C05458=1080.176,351.466,404.288,176.034,28.029,154.818
C05459=1080.171,351.219,404.324,176.031,28.024,154.817
C05460=1080.164,350.972,404.359,176.028,28.019,154.816
C05461=1080.158,350.724,404.394,176.025,28.013,154.815
C05462=1080.153,350.477,404.429,176.022,28.008,154.814
C05463=1080.146,350.229,404.464,176.018,28.002,154.813
C05464=1080.140,349.982,404.500,176.015,27.997,154.812
C05465=1080.134,349.735,404.535,176.012,27.992,154.811
C05466=1080.128,349.487,404.570,176.009,27.987,154.810
C05467=1080.121,349.239,404.605,176.005,27.981,154.809
C05468=1080.116,348.992,404.640,176.002,27.976,154.808
C05469=1080.109,348.745,404.675,175.999,27.971,154.807
C05470=1080.103,348.497,404.710,175.995,27.965,154.807
C05471=1080.097,348.250,404.745,175.992,27.960,154.806
C05472=1080.091,348.002,404.781,175.989,27.955,154.805
C05473=1080.085,347.755,404.815,175.985,27.950,154.804
C05474=1080.079,347.507,404.851,175.982,27.944,154.803
C05475=1080.073,347.259,404.885,175.979,27.939,154.802
C05476=1080.067,347.012,404.920,175.976,27.934,154.801
C05477=1080.061,346.765,404.956,175.973,27.929,154.800
C05478=1080.055,346.518,404.990,175.970,27.924,154.799
C05479=1080.049,346.270,405.025,175.966,27.918,154.798
C05480=1080.043,346.022,405.060,175.963,27.913,154.797
C05481=1080.037,345.775,405.095,175.959,27.908,154.797
C05482=1080.030,345.527,405.130,175.956,27.903,154.796
C05483=1080.025,345.280,405.165,175.953,27.898,154.795
C05484=1080.018,345.032,405.199,175.950,27.893,154.794
C05485=1080.009,344.621,405.257,175.945,27.884,154.793
C05486=1079.998,344.208,405.314,175.939,27.876,154.791
C05487=1079.988,343.795,405.372,175.934,27.867,154.790
C05488=1079.978,343.384,405.430,175.928,27.858,154.788
C05489=1079.972,343.135,405.465,175.925,27.854,154.787
C05490=1079.967,342.888,405.499,175.922,27.848,154.786
C05491=1079.960,342.641,405.534,175.919,27.843,154.786
C05492=1079.954,342.394,405.568,175.916,27.839,154.785
C05493=1079.947,342.146,405.603,175.912,27.833,154.784
C05494=1079.942,341.898,405.637,175.909,27.828,154.783
C05495=1079.936,341.650,405.672,175.906,27.823,154.782
C05496=1079.930,341.403,405.706,175.903,27.818,154.781
C05497=1079.923,341.155,405.741,175.899,27.813,154.781
C05498=1079.917,340.908,405.775,175.896,27.808,154.780
C05499=1079.912,340.661,405.809,175.893,27.803,154.779
C05500=1079.906,340.412,405.844,175.890,27.798,154.778
C05501=1079.900,340.165,405.878,175.887,27.793,154.777
C05502=1079.894,339.917,405.913,175.884,27.788,154.776
C05503=1079.888,339.670,405.947,175.881,27.784,154.775
C05504=1079.882,339.423,405.981,175.877,27.778,154.775
C05505=1079.875,339.175,406.015,175.874,27.773,154.774
C05506=1079.869,338.927,406.049,175.871,27.768,154.773
C05507=1079.864,338.679,406.084,175.867,27.763,154.772
C05508=1079.858,338.432,406.118,175.864,27.758,154.771
C05509=1079.852,338.184,406.152,175.861,27.754,154.770
C05510=1079.846,337.936,406.187,175.858,27.748,154.770
C05511=1079.840,337.689,406.221,175.855,27.744,154.769
C05512=1079.834,337.441,406.254,175.852,27.739,154.768
C05513=1079.828,337.193,406.288,175.849,27.734,154.767
C05514=1079.822,336.946,406.322,175.846,27.729,154.766
C05515=1079.816,336.699,406.357,175.843,27.724,154.766
C05516=1079.809,336.451,406.391,175.839,27.720,154.765
C05517=1079.804,336.203,406.425,175.836,27.715,154.764
C05518=1079.797,335.956,406.458,175.833,27.710,154.763
C05519=1079.791,335.708,406.492,175.830,27.705,154.762
C05520=1079.785,335.461,406.526,175.827,27.700,154.762
C05521=1079.779,335.213,406.560,175.824,27.695,154.761
C05522=1079.773,334.965,406.594,175.821,27.691,154.760
C05523=1079.767,334.717,406.628,175.818,27.685,154.759
C05524=1079.761,334.470,406.662,175.815,27.681,154.758
C05525=1079.756,334.222,406.695,175.811,27.676,154.758
C05526=1079.749,333.974,406.730,175.807,27.671,154.757
C05527=1079.744,333.726,406.763,175.804,27.666,154.756
C05528=1079.737,333.479,406.797,175.801,27.662,154.755
C05529=1079.731,333.232,406.831,175.798,27.656,154.754
C05530=1079.726,332.984,406.864,175.795,27.652,154.754
C05531=1079.719,332.736,406.898,175.792,27.647,154.753
C05532=1079.714,332.488,406.932,175.789,27.642,154.752
C05533=1079.708,332.241,406.966,175.786,27.638,154.751
C05534=1079.702,331.993,406.999,175.783,27.633,154.750
C05535=1079.696,331.746,407.033,175.780,27.628,154.750
C05536=1079.690,331.498,407.066,175.777,27.624,154.749
C05537=1079.679,331.080,407.123,175.772,27.615,154.748
C05538=1079.669,330.662,407.179,175.766,27.608,154.746
C05539=1079.659,330.245,407.235,175.760,27.600,154.745
C05540=1079.648,329.827,407.292,175.756,27.592,154.744
C05541=1079.642,329.579,407.326,175.753,27.588,154.743
C05542=1079.636,329.331,407.358,175.750,27.583,154.742
C05543=1079.630,329.084,407.392,175.746,27.579,154.742
C05544=1079.624,328.836,407.425,175.743,27.574,154.741
C05545=1079.618,328.588,407.458,175.740,27.569,154.740
C05546=1079.612,328.341,407.491,175.737,27.565,154.739
C05547=1079.606,328.092,407.525,175.734,27.560,154.739
C05548=1079.599,327.845,407.558,175.731,27.555,154.738
C05549=1079.594,327.597,407.592,175.728,27.551,154.737
C05550=1079.587,327.350,407.624,175.725,27.546,154.736
C05551=1079.582,327.102,407.658,175.721,27.542,154.736
C05552=1079.575,326.854,407.690,175.718,27.537,154.735
C05553=1079.570,326.606,407.724,175.715,27.533,154.734
C05554=1079.564,326.359,407.757,175.712,27.528,154.733
C05555=1079.558,326.112,407.791,175.709,27.523,154.733
C05556=1079.551,325.863,407.824,175.707,27.519,154.732
C05557=1079.545,325.615,407.857,175.704,27.515,154.731
C05558=1079.539,325.368,407.890,175.700,27.510,154.730
C05559=1079.533,325.120,407.923,175.697,27.506,154.730
C05560=1079.527,324.872,407.956,175.694,27.501,154.729
C05561=1079.521,324.625,407.989,175.691,27.497,154.728
C05562=1079.515,324.377,408.022,175.688,27.492,154.728
C05563=1079.509,324.129,408.055,175.685,27.487,154.727
C05564=1079.503,323.881,408.088,175.682,27.483,154.726
C05565=1079.497,323.633,408.120,175.678,27.478,154.725
C05566=1079.491,323.385,408.153,175.676,27.474,154.725
C05567=1079.486,323.138,408.186,175.673,27.469,154.724
C05568=1079.479,322.890,408.219,175.670,27.465,154.723
C05569=1079.474,322.642,408.252,175.667,27.460,154.723
C05570=1079.467,322.394,408.285,175.664,27.456,154.722
C05571=1079.461,322.147,408.318,175.660,27.451,154.721
C05572=1079.457,321.899,408.350,175.657,27.447,154.720
C05573=1079.450,321.651,408.383,175.654,27.442,154.720
C05574=1079.445,321.404,408.416,175.651,27.438,154.719
C05575=1079.438,321.156,408.449,175.649,27.434,154.718
C05576=1079.432,320.908,408.482,175.646,27.429,154.717
C05577=1079.427,320.660,408.514,175.643,27.425,154.717
C05578=1079.421,320.412,408.547,175.639,27.420,154.716
C05579=1079.414,320.165,408.580,175.636,27.416,154.715
C05580=1079.409,319.916,408.612,175.633,27.411,154.715
C05581=1079.403,319.669,408.645,175.630,27.407,154.714
C05582=1079.397,319.422,408.677,175.628,27.402,154.713
C05583=1079.392,319.173,408.710,175.625,27.398,154.713
C05584=1079.386,318.925,408.743,175.622,27.393,154.712
C05585=1079.379,318.678,408.775,175.618,27.389,154.711
C05586=1079.374,318.430,408.807,175.615,27.384,154.710
C05587=1079.368,318.182,408.840,175.612,27.380,154.710
C05588=1079.362,317.934,408.872,175.610,27.376,154.709
C05589=1079.357,317.723,408.901,175.607,27.372,154.708
C05590=1079.353,317.510,408.928,175.605,27.368,154.708
C05591=1079.347,317.297,408.956,175.602,27.364,154.707
C05592=1079.342,317.086,408.985,175.599,27.360,154.707
C05593=1079.337,316.874,409.012,175.597,27.356,154.706
C05594=1079.332,316.662,409.039,175.594,27.353,154.705
C05595=1079.328,316.449,409.067,175.592,27.349,154.705
C05596=1079.323,316.238,409.095,175.589,27.345,154.704
C05597=1079.317,315.989,409.127,175.587,27.341,154.703
C05598=1079.311,315.741,409.159,175.584,27.337,154.703
C05599=1079.306,315.494,409.192,175.580,27.332,154.702
C05600=1079.300,315.246,409.224,175.577,27.327,154.701
C05601=1079.294,314.998,409.257,175.574,27.323,154.701
C05602=1079.288,314.751,409.289,175.572,27.319,154.700
C05603=1079.282,314.502,409.321,175.569,27.314,154.699
C05604=1079.276,314.255,409.354,175.566,27.310,154.699
C05605=1079.270,314.007,409.386,175.562,27.306,154.698
C05606=1079.264,313.758,409.418,175.559,27.302,154.697
C05607=1079.258,313.511,409.449,175.556,27.297,154.697
C05608=1079.251,313.264,409.481,175.554,27.293,154.696
C05609=1079.245,313.015,409.513,175.551,27.289,154.695
C05610=1079.239,312.767,409.545,175.548,27.285,154.695
C05611=1079.233,312.519,409.578,175.544,27.281,154.694
C05612=1079.228,312.272,409.609,175.541,27.276,154.694
C05613=1079.221,312.024,409.641,175.539,27.272,154.693
C05614=1079.215,311.776,409.673,175.536,27.268,154.692
C05615=1079.210,311.529,409.705,175.533,27.264,154.692
C05616=1079.204,311.280,409.737,175.530,27.260,154.691
C05617=1079.198,311.032,409.769,175.527,27.256,154.690
C05618=1079.191,310.784,409.800,175.524,27.251,154.690
C05619=1079.186,310.537,409.832,175.521,27.247,154.689
C05620=1079.180,310.288,409.864,175.518,27.243,154.688
C05621=1079.174,310.040,409.896,175.515,27.238,154.688
C05622=1079.168,309.793,409.927,175.512,27.234,154.687
C05623=1079.162,309.545,409.959,175.509,27.230,154.686
C05624=1079.156,309.297,409.991,175.506,27.226,154.686
C05625=1079.150,309.049,410.023,175.503,27.222,154.685
C05626=1079.143,308.801,410.054,175.501,27.218,154.684
C05627=1079.138,308.554,410.086,175.498,27.213,154.684
C05628=1079.132,308.305,410.118,175.494,27.209,154.683
C05629=1079.127,308.058,410.150,175.491,27.205,154.682
C05630=1079.120,307.810,410.181,175.488,27.201,154.682
C05631=1079.114,307.562,410.213,175.486,27.197,154.681
C05632=1079.109,307.314,410.245,175.483,27.193,154.681
C05633=1079.102,307.066,410.276,175.480,27.188,154.680
C05634=1079.096,306.819,410.308,175.476,27.184,154.679
C05635=1079.091,306.570,410.339,175.474,27.180,154.679
C05636=1079.085,306.323,410.370,175.471,27.176,154.678
C05637=1079.079,306.075,410.402,175.468,27.172,154.677
C05638=1079.073,305.827,410.434,175.465,27.167,154.677
C05639=1079.067,305.579,410.465,175.463,27.163,154.676
C05640=1079.061,305.331,410.496,175.459,27.159,154.675
C05641=1079.056,305.083,410.528,175.456,27.155,154.675
C05642=1079.049,304.836,410.560,175.454,27.151,154.674
C05643=1079.043,304.587,410.592,175.451,27.147,154.674
C05644=1079.038,304.339,410.622,175.448,27.143,154.673
C05645=1079.032,304.129,410.649,175.445,27.139,154.672
C05646=1079.028,303.919,410.676,175.443,27.136,154.672
C05647=1079.023,303.708,410.703,175.441,27.132,154.671
C05648=1079.018,303.497,410.729,175.437,27.128,154.671
C05649=1079.013,303.287,410.756,175.435,27.125,154.670
C05650=1079.008,303.076,410.783,175.433,27.121,154.670
C05651=1079.003,302.866,410.808,175.431,27.118,154.669
C05652=1078.998,302.655,410.836,175.428,27.115,154.669
C05653=1078.993,302.407,410.867,175.425,27.110,154.668
C05654=1078.986,302.159,410.898,175.422,27.106,154.667
C05655=1078.981,301.911,410.929,175.420,27.102,154.667
C05656=1078.975,301.663,410.960,175.417,27.098,154.666
C05657=1078.970,301.415,410.991,175.413,27.094,154.666
C05658=1078.964,301.167,411.023,175.411,27.090,154.665
C05659=1078.958,300.919,411.054,175.408,27.086,154.664
C05660=1078.952,300.671,411.085,175.405,27.081,154.664
C05661=1078.947,300.423,411.116,175.403,27.077,154.663
C05662=1078.941,300.175,411.148,175.400,27.073,154.662
C05663=1078.935,299.927,411.178,175.396,27.069,154.662
C05664=1078.929,299.680,411.210,175.394,27.065,154.661
C05665=1078.923,299.431,411.241,175.391,27.061,154.661
C05666=1078.918,299.184,411.272,175.388,27.057,154.660
C05667=1078.912,298.936,411.303,175.385,27.052,154.659
C05668=1078.907,298.688,411.334,175.383,27.048,154.659
C05669=1078.901,298.440,411.366,175.379,27.044,154.658
C05670=1078.895,298.192,411.396,175.377,27.040,154.657
C05671=1078.890,297.944,411.427,175.374,27.036,154.657
C05672=1078.884,297.697,411.458,175.371,27.032,154.656
C05673=1078.877,297.448,411.489,175.369,27.028,154.656
C05674=1078.872,297.200,411.520,175.365,27.024,154.655
C05675=1078.866,296.952,411.550,175.362,27.020,154.654
C05676=1078.860,296.704,411.581,175.360,27.016,154.654
C05677=1078.855,296.456,411.612,175.357,27.012,154.653
C05678=1078.849,296.208,411.643,175.354,27.008,154.652
C05679=1078.842,295.960,411.673,175.351,27.004,154.652
C05680=1078.836,295.712,411.704,175.348,27.000,154.651
C05681=1078.831,295.464,411.735,175.345,26.996,154.651
C05682=1078.825,295.215,411.765,175.343,26.992,154.650
C05683=1078.819,294.968,411.796,175.340,26.988,154.649
C05684=1078.813,294.720,411.827,175.337,26.984,154.649
C05685=1078.807,294.472,411.857,175.334,26.980,154.648
C05686=1078.802,294.224,411.888,175.331,26.976,154.648
C05687=1078.796,293.976,411.919,175.328,26.972,154.647
C05688=1078.790,293.728,411.949,175.326,26.968,154.647
C05689=1078.784,293.480,411.980,175.323,26.964,154.646
C05690=1078.778,293.232,412.010,175.320,26.960,154.645
C05691=1078.772,292.984,412.041,175.317,26.956,154.645
C05692=1078.766,292.736,412.071,175.314,26.952,154.644
C05693=1078.761,292.488,412.102,175.312,26.948,154.644
C05694=1078.755,292.240,412.132,175.309,26.944,154.643
C05695=1078.749,291.991,412.163,175.306,26.940,154.642
C05696=1078.743,291.744,412.193,175.303,26.936,154.642
C05697=1078.737,291.496,412.224,175.300,26.932,154.641
C05698=1078.732,291.247,412.253,175.298,26.928,154.641
C05699=1078.726,291.000,412.284,175.295,26.924,154.640
C05700=1078.719,290.751,412.314,175.292,26.920,154.639
C05701=1078.710,290.344,412.364,175.288,26.914,154.639
C05702=1078.700,289.938,412.414,175.283,26.907,154.638
C05703=1078.691,289.531,412.464,175.279,26.901,154.637
C05704=1078.682,289.124,412.513,175.274,26.894,154.636
C05705=1078.675,288.876,412.544,175.271,26.891,154.635
C05706=1078.670,288.628,412.573,175.268,26.887,154.635
C05707=1078.664,288.380,412.604,175.265,26.883,154.634
C05708=1078.658,288.132,412.634,175.262,26.879,154.633
C05709=1078.652,287.884,412.663,175.260,26.875,154.633
C05710=1078.646,287.636,412.693,175.257,26.871,154.632
C05711=1078.640,287.388,412.724,175.254,26.868,154.632
C05712=1078.634,287.139,412.754,175.251,26.863,154.631
C05713=1078.628,286.891,412.784,175.249,26.860,154.631
C05714=1078.623,286.643,412.814,175.246,26.856,154.630
C05715=1078.617,286.395,412.844,175.243,26.852,154.629
C05716=1078.611,286.147,412.874,175.240,26.848,154.629
C05717=1078.605,285.899,412.903,175.237,26.844,154.628
C05718=1078.599,285.651,412.934,175.235,26.840,154.628
C05719=1078.594,285.403,412.963,175.232,26.836,154.627
C05720=1078.588,285.155,412.994,175.230,26.832,154.627
C05721=1078.582,284.906,413.023,175.226,26.828,154.626
C05722=1078.577,284.659,413.054,175.224,26.825,154.625
C05723=1078.570,284.410,413.083,175.221,26.821,154.625
C05724=1078.564,284.163,413.113,175.218,26.817,154.624
C05725=1078.559,283.914,413.143,175.216,26.813,154.624
C05726=1078.553,283.666,413.173,175.213,26.809,154.623
C05727=1078.548,283.418,413.203,175.210,26.805,154.623
C05728=1078.541,283.170,413.233,175.207,26.801,154.622
C05729=1078.536,282.922,413.262,175.205,26.798,154.621
C05730=1078.530,282.674,413.292,175.202,26.794,154.621
C05731=1078.524,282.426,413.322,175.200,26.790,154.620
C05732=1078.519,282.177,413.352,175.196,26.786,154.620
C05733=1078.513,281.929,413.381,175.194,26.782,154.619
C05734=1078.507,281.681,413.411,175.191,26.778,154.619
C05735=1078.501,281.433,413.441,175.189,26.774,154.618
C05736=1078.496,281.184,413.471,175.186,26.770,154.617
C05737=1078.489,280.937,413.500,175.182,26.766,154.617
C05738=1078.484,280.688,413.530,175.180,26.763,154.616
C05739=1078.478,280.440,413.560,175.177,26.758,154.616
C05740=1078.472,280.192,413.589,175.175,26.755,154.615
C05741=1078.466,279.943,413.618,175.172,26.751,154.615
C05742=1078.460,279.696,413.648,175.169,26.747,154.614
C05743=1078.454,279.447,413.678,175.166,26.743,154.614
C05744=1078.449,279.199,413.707,175.164,26.740,154.613
C05745=1078.442,278.951,413.736,175.161,26.736,154.613
C05746=1078.437,278.702,413.766,175.159,26.732,154.612
C05747=1078.431,278.454,413.795,175.155,26.728,154.611
C05748=1078.425,278.206,413.825,175.153,26.724,154.611
C05749=1078.420,277.959,413.855,175.150,26.720,154.610
C05750=1078.414,277.711,413.884,175.148,26.717,154.610
C05751=1078.408,277.462,413.913,175.145,26.713,154.609
C05752=1078.402,277.214,413.942,175.142,26.709,154.609
C05753=1078.393,276.817,413.989,175.138,26.703,154.608
C05754=1078.384,276.419,414.036,175.134,26.697,154.607
C05755=1078.374,276.023,414.083,175.129,26.691,154.606
C05756=1078.365,275.626,414.130,175.125,26.685,154.605
C05757=1078.359,275.378,414.159,175.122,26.681,154.605
C05758=1078.353,275.130,414.188,175.120,26.677,154.604
C05759=1078.347,274.881,414.218,175.117,26.673,154.603
C05760=1078.341,274.633,414.247,175.115,26.670,154.603
C05761=1078.337,274.385,414.275,175.112,26.666,154.602
C05762=1078.330,274.137,414.304,175.109,26.662,154.602
C05763=1078.325,273.888,414.334,175.106,26.658,154.601
C05764=1078.319,273.640,414.363,175.104,26.654,154.601
C05765=1078.312,273.392,414.392,175.101,26.651,154.600
C05766=1078.307,273.144,414.421,175.099,26.647,154.600
C05767=1078.301,272.896,414.450,175.095,26.643,154.599
C05768=1078.296,272.647,414.479,175.093,26.639,154.599
C05769=1078.290,272.399,414.508,175.090,26.635,154.598
C05770=1078.283,272.151,414.537,175.088,26.632,154.597
C05771=1078.278,271.903,414.565,175.085,26.628,154.597
C05772=1078.273,271.654,414.595,175.082,26.624,154.596
C05773=1078.266,271.406,414.624,175.080,26.621,154.596
C05774=1078.260,271.157,414.652,175.077,26.617,154.595
C05775=1078.255,270.909,414.682,175.075,26.613,154.595
C05776=1078.249,270.662,414.711,175.072,26.609,154.594
C05777=1078.243,270.413,414.739,175.069,26.605,154.594
C05778=1078.238,270.164,414.769,175.066,26.602,154.593
C05779=1078.232,269.916,414.798,175.064,26.598,154.593
C05780=1078.226,269.668,414.826,175.061,26.594,154.592
C05781=1078.220,269.420,414.855,175.059,26.591,154.592
C05782=1078.214,269.172,414.884,175.056,26.587,154.591
C05783=1078.209,268.924,414.912,175.053,26.583,154.590
C05784=1078.203,268.675,414.941,175.051,26.579,154.590
C05785=1078.197,268.427,414.970,175.048,26.575,154.589
C05786=1078.191,268.179,414.999,175.046,26.572,154.589
C05787=1078.185,267.930,415.027,175.042,26.568,154.588
C05788=1078.179,267.682,415.056,175.040,26.564,154.588
C05789=1078.174,267.433,415.084,175.037,26.561,154.587
C05790=1078.168,267.186,415.113,175.035,26.557,154.587
C05791=1078.162,266.937,415.141,175.033,26.553,154.586
C05792=1078.156,266.689,415.171,175.029,26.550,154.586
C05793=1078.151,266.441,415.198,175.027,26.545,154.585
C05794=1078.145,266.192,415.227,175.024,26.542,154.585
C05795=1078.138,265.944,415.256,175.022,26.538,154.584
C05796=1078.133,265.696,415.284,175.020,26.535,154.584
C05797=1078.128,265.447,415.313,175.016,26.531,154.583
C05798=1078.122,265.199,415.342,175.014,26.527,154.583
C05799=1078.116,264.951,415.370,175.011,26.523,154.582
C05800=1078.110,264.703,415.399,175.009,26.520,154.581
C05801=1078.104,264.454,415.427,175.007,26.516,154.581
C05802=1078.099,264.206,415.455,175.004,26.512,154.580
C05803=1078.093,263.957,415.483,175.001,26.508,154.580
C05804=1078.087,263.710,415.512,174.998,26.504,154.579
C05805=1078.077,263.315,415.557,174.994,26.499,154.579
C05806=1078.068,262.921,415.601,174.991,26.493,154.578
C05807=1078.059,262.527,415.646,174.986,26.487,154.577
C05808=1078.049,262.134,415.691,174.982,26.481,154.576
C05809=1078.043,261.885,415.719,174.979,26.478,154.576
C05810=1078.038,261.637,415.747,174.977,26.474,154.575
C05811=1078.031,261.389,415.775,174.974,26.470,154.575
C05812=1078.025,261.140,415.803,174.971,26.467,154.574
C05813=1078.020,260.892,415.832,174.969,26.463,154.573
C05814=1078.014,260.644,415.860,174.966,26.459,154.573
C05815=1078.008,260.396,415.888,174.964,26.456,154.573
C05816=1078.002,260.147,415.916,174.961,26.453,154.572
C05817=1077.996,259.898,415.944,174.958,26.449,154.572
C05818=1077.990,259.650,415.972,174.956,26.445,154.571
C05819=1077.984,259.402,416.001,174.954,26.442,154.570
C05820=1077.978,259.154,416.028,174.951,26.438,154.570
C05821=1077.972,258.905,416.056,174.948,26.434,154.569
C05822=1077.967,258.657,416.084,174.945,26.430,154.569
C05823=1077.961,258.408,416.113,174.943,26.427,154.568
C05824=1077.955,258.161,416.140,174.941,26.423,154.568
C05825=1077.949,257.912,416.168,174.938,26.419,154.567
C05826=1077.944,257.664,416.196,174.935,26.416,154.567
C05827=1077.938,257.415,416.225,174.933,26.412,154.566
C05828=1077.932,257.167,416.251,174.930,26.408,154.566
C05829=1077.926,256.918,416.280,174.928,26.405,154.565
C05830=1077.921,256.670,416.308,174.926,26.401,154.565
C05831=1077.915,256.421,416.336,174.922,26.397,154.564
C05832=1077.909,256.173,416.363,174.920,26.394,154.564
C05833=1077.903,255.925,416.392,174.918,26.390,154.563
C05834=1077.898,255.677,416.420,174.915,26.386,154.563
C05835=1077.891,255.428,416.447,174.913,26.383,154.562
C05836=1077.886,255.179,416.475,174.910,26.379,154.562
C05837=1077.880,254.931,416.503,174.907,26.375,154.561
C05838=1077.874,254.683,416.530,174.905,26.372,154.561
C05839=1077.868,254.434,416.558,174.903,26.368,154.560
C05840=1077.863,254.186,416.586,174.900,26.364,154.560
C05841=1077.857,253.938,416.613,174.897,26.360,154.559
C05842=1077.851,253.689,416.642,174.895,26.357,154.559
C05843=1077.846,253.440,416.669,174.892,26.353,154.558
C05844=1077.839,253.192,416.696,174.890,26.349,154.557
C05845=1077.834,252.944,416.724,174.888,26.346,154.557
C05846=1077.829,252.695,416.752,174.885,26.342,154.556
C05847=1077.822,252.447,416.779,174.882,26.338,154.556
C05848=1077.817,252.199,416.807,174.880,26.335,154.555
C05849=1077.812,251.950,416.835,174.877,26.331,154.555
C05850=1077.805,251.702,416.862,174.875,26.327,154.554
C05851=1077.800,251.453,416.890,174.873,26.324,154.554
C05852=1077.795,251.205,416.918,174.869,26.320,154.553
C05853=1077.788,250.956,416.945,174.867,26.316,154.553
C05854=1077.783,250.708,416.973,174.865,26.313,154.552
C05855=1077.777,250.460,417.000,174.862,26.309,154.552
C05856=1077.771,250.211,417.027,174.860,26.305,154.551
C05857=1077.763,249.815,417.072,174.856,26.299,154.550
C05858=1077.753,249.418,417.115,174.852,26.293,154.549
C05859=1077.744,249.021,417.159,174.848,26.287,154.549
C05860=1077.735,248.625,417.202,174.844,26.281,154.548
C05861=1077.729,248.376,417.230,174.842,26.278,154.547
C05862=1077.724,248.128,417.257,174.840,26.274,154.547
C05863=1077.718,247.880,417.285,174.836,26.270,154.546
C05864=1077.713,247.631,417.312,174.834,26.267,154.546
C05865=1077.707,247.382,417.339,174.832,26.263,154.545
C05866=1077.701,247.134,417.367,174.829,26.259,154.545
C05867=1077.696,246.886,417.394,174.827,26.255,154.544
C05868=1077.690,246.637,417.421,174.825,26.252,154.544
C05869=1077.684,246.389,417.449,174.822,26.248,154.543
C05870=1077.678,246.140,417.475,174.819,26.244,154.543
C05871=1077.673,245.892,417.503,174.817,26.241,154.542
C05872=1077.667,245.644,417.530,174.815,26.237,154.542
C05873=1077.661,245.395,417.557,174.813,26.234,154.541
C05874=1077.656,245.146,417.584,174.809,26.230,154.541
C05875=1077.650,244.898,417.611,174.807,26.226,154.540
C05876=1077.644,244.650,417.638,174.805,26.223,154.539
C05877=1077.639,244.401,417.666,174.802,26.219,154.539
C05878=1077.632,244.152,417.693,174.800,26.215,154.538
C05879=1077.627,243.904,417.719,174.798,26.211,154.538
C05880=1077.622,243.655,417.747,174.795,26.208,154.537
C05881=1077.616,243.407,417.773,174.792,26.204,154.537
C05882=1077.610,243.159,417.801,174.790,26.200,154.536
C05883=1077.604,242.910,417.828,174.788,26.197,154.536
C05884=1077.598,242.661,417.855,174.786,26.193,154.535
C05885=1077.593,242.413,417.881,174.783,26.189,154.535
C05886=1077.587,242.165,417.908,174.780,26.186,154.534
C05887=1077.581,241.916,417.935,174.778,26.183,154.534
C05888=1077.575,241.667,417.962,174.776,26.179,154.533
C05889=1077.570,241.419,417.989,174.773,26.175,154.533
C05890=1077.564,241.170,418.016,174.771,26.171,154.532
C05891=1077.558,240.922,418.042,174.768,26.168,154.532
C05892=1077.552,240.674,418.069,174.766,26.164,154.531
C05893=1077.547,240.425,418.096,174.763,26.160,154.531
C05894=1077.540,240.176,418.123,174.761,26.157,154.530
C05895=1077.534,239.928,418.149,174.759,26.153,154.530
C05896=1077.529,239.679,418.176,174.756,26.150,154.529
C05897=1077.524,239.431,418.203,174.754,26.146,154.529
C05898=1077.518,239.182,418.230,174.751,26.142,154.528
C05899=1077.512,238.934,418.256,174.749,26.139,154.528
C05900=1077.506,238.685,418.283,174.747,26.135,154.527
C05901=1077.500,238.437,418.310,174.744,26.132,154.527
C05902=1077.494,238.188,418.337,174.741,26.128,154.526
C05903=1077.489,237.939,418.363,174.739,26.124,154.526
C05904=1077.483,237.691,418.389,174.737,26.121,154.525
C05905=1077.477,237.443,418.416,174.735,26.117,154.525
C05906=1077.471,237.194,418.443,174.733,26.113,154.524
C05907=1077.466,236.946,418.469,174.729,26.110,154.524
C05908=1077.460,236.698,418.496,174.727,26.106,154.523
C05909=1077.450,236.293,418.539,174.724,26.100,154.522
C05910=1077.441,235.891,418.582,174.720,26.094,154.521
C05911=1077.432,235.487,418.624,174.715,26.088,154.521
C05912=1077.423,235.085,418.667,174.712,26.082,154.520
C05913=1077.417,234.836,418.694,174.709,26.079,154.519
C05914=1077.412,234.587,418.720,174.707,26.075,154.519
C05915=1077.406,234.339,418.747,174.705,26.071,154.518
C05916=1077.400,234.091,418.773,174.703,26.068,154.518
C05917=1077.395,233.842,418.799,174.700,26.064,154.517
C05918=1077.389,233.593,418.826,174.698,26.060,154.517
C05919=1077.383,233.345,418.853,174.695,26.057,154.516
C05920=1077.377,233.095,418.879,174.693,26.053,154.516
C05921=1077.371,232.847,418.906,174.691,26.050,154.515
C05922=1077.366,232.598,418.931,174.688,26.046,154.515
C05923=1077.360,232.350,418.957,174.686,26.042,154.514
C05924=1077.354,232.102,418.984,174.684,26.039,154.514
C05925=1077.349,231.853,419.010,174.681,26.035,154.513
C05926=1077.343,231.605,419.036,174.679,26.032,154.513
C05927=1077.337,231.356,419.062,174.676,26.028,154.512
C05928=1077.332,231.107,419.089,174.674,26.024,154.512
C05929=1077.326,230.858,419.115,174.672,26.020,154.511
C05930=1077.320,230.610,419.141,174.670,26.017,154.511
C05931=1077.314,230.361,419.167,174.667,26.013,154.510
C05932=1077.308,230.113,419.193,174.665,26.010,154.510
C05933=1077.303,229.864,419.219,174.662,26.006,154.509
C05934=1077.296,229.616,419.245,174.660,26.002,154.509
C05935=1077.291,229.367,419.271,174.658,25.998,154.508
C05936=1077.285,229.118,419.297,174.656,25.995,154.508
C05937=1077.279,228.870,419.323,174.653,25.992,154.507
C05938=1077.273,228.621,419.349,174.651,25.988,154.507
C05939=1077.268,228.372,419.375,174.648,25.984,154.506
C05940=1077.261,228.124,419.401,174.646,25.981,154.506
C05941=1077.256,227.875,419.427,174.644,25.977,154.505
C05942=1077.251,227.626,419.453,174.642,25.973,154.504
C05943=1077.245,227.379,419.479,174.639,25.970,154.504
C05944=1077.239,227.130,419.505,174.637,25.966,154.503
C05945=1077.234,226.881,419.531,174.635,25.963,154.503
C05946=1077.227,226.633,419.557,174.632,25.959,154.503
C05947=1077.222,226.384,419.583,174.630,25.955,154.502
C05948=1077.215,226.135,419.608,174.628,25.952,154.502
C05949=1077.210,225.886,419.634,174.625,25.948,154.501
C05950=1077.204,225.638,419.661,174.623,25.945,154.500
C05951=1077.199,225.390,419.686,174.621,25.941,154.500
C05952=1077.193,225.141,419.712,174.619,25.937,154.499
C05953=1077.187,224.892,419.737,174.616,25.933,154.499
C05954=1077.182,224.643,419.763,174.614,25.930,154.498
C05955=1077.176,224.395,419.789,174.611,25.926,154.498
C05956=1077.170,224.146,419.815,174.609,25.922,154.497
C05957=1077.165,223.898,419.840,174.607,25.919,154.497
C05958=1077.158,223.649,419.866,174.605,25.915,154.496
C05959=1077.153,223.400,419.892,174.603,25.912,154.496
C05960=1077.148,223.151,419.918,174.601,25.908,154.495
C05961=1077.138,222.740,419.960,174.596,25.902,154.494
C05962=1077.129,222.328,420.002,174.592,25.896,154.494
C05963=1077.119,221.917,420.044,174.589,25.890,154.493
C05964=1077.110,221.506,420.087,174.585,25.884,154.492
C05965=1077.104,221.257,420.112,174.583,25.881,154.491
C05966=1077.098,221.008,420.138,174.581,25.877,154.491
C05967=1077.092,220.759,420.164,174.579,25.873,154.490
C05968=1077.086,220.510,420.189,174.577,25.870,154.490
C05969=1077.081,220.262,420.214,174.573,25.866,154.489
C05970=1077.075,220.013,420.240,174.571,25.862,154.489
C05971=1077.069,219.765,420.265,174.569,25.858,154.488
C05972=1077.063,219.516,420.291,174.567,25.855,154.488
C05973=1077.058,219.268,420.316,174.565,25.851,154.487
C05974=1077.052,219.019,420.342,174.563,25.848,154.487
C05975=1077.045,218.770,420.367,174.560,25.844,154.486
C05976=1077.040,218.521,420.392,174.558,25.841,154.486
C05977=1077.035,218.273,420.417,174.556,25.837,154.485
C05978=1077.028,218.024,420.442,174.554,25.833,154.485
C05979=1077.023,217.775,420.468,174.551,25.830,154.484
C05980=1077.017,217.527,420.493,174.549,25.826,154.484
C05981=1077.011,217.279,420.519,174.547,25.822,154.483
C05982=1077.006,217.029,420.544,174.544,25.819,154.483
C05983=1077.000,216.780,420.569,174.542,25.815,154.482
C05984=1076.994,216.532,420.594,174.540,25.811,154.482
C05985=1076.988,216.284,420.620,174.538,25.808,154.481
C05986=1076.983,216.034,420.645,174.536,25.804,154.481
C05987=1076.977,215.786,420.670,174.534,25.800,154.480
C05988=1076.971,215.537,420.695,174.532,25.797,154.480
C05989=1076.966,215.289,420.721,174.529,25.793,154.479
C05990=1076.960,215.040,420.745,174.527,25.790,154.479
C05991=1076.954,214.791,420.771,174.525,25.786,154.478
C05992=1076.948,214.543,420.796,174.522,25.782,154.478
C05993=1076.943,214.294,420.821,174.520,25.778,154.477
C05994=1076.937,214.045,420.846,174.518,25.775,154.477
C05995=1076.931,213.797,420.871,174.516,25.771,154.476
C05996=1076.926,213.548,420.896,174.513,25.767,154.475
C05997=1076.921,213.299,420.921,174.511,25.764,154.475
C05998=1076.914,213.051,420.947,174.509,25.760,154.474
C05999=1076.909,212.801,420.971,174.507,25.757,154.474
C06000=1076.903,212.553,420.996,174.505,25.753,154.474
C06001=1076.897,212.304,421.021,174.503,25.750,154.473
C06002=1076.891,212.056,421.046,174.501,25.746,154.472
C06003=1076.886,211.807,421.070,174.498,25.742,154.472
C06004=1076.879,211.558,421.096,174.496,25.739,154.471
C06005=1076.875,211.309,421.121,174.494,25.735,154.471
C06006=1076.869,211.061,421.146,174.492,25.731,154.470
C06007=1076.863,210.812,421.170,174.490,25.728,154.470
C06008=1076.857,210.563,421.196,174.488,25.724,154.469
C06009=1076.852,210.315,421.220,174.486,25.720,154.469
C06010=1076.846,210.066,421.245,174.483,25.717,154.468
C06011=1076.840,209.817,421.270,174.480,25.713,154.468
C06012=1076.834,209.569,421.295,174.478,25.709,154.467
C06013=1076.825,209.161,421.335,174.475,25.703,154.466
C06014=1076.816,208.754,421.376,174.472,25.698,154.466
C06015=1076.806,208.347,421.416,174.468,25.692,154.465
C06016=1076.796,207.939,421.457,174.465,25.686,154.464
C06017=1076.773,206.902,421.557,174.351,25.626,154.464
C06018=1076.768,206.653,421.581,174.349,25.623,154.464
C06019=1076.761,206.404,421.605,174.347,25.620,154.464
C06020=1076.756,206.156,421.630,174.344,25.618,154.464
C06021=1076.750,205.907,421.654,174.343,25.615,154.463
C06022=1076.745,205.658,421.677,174.341,25.613,154.463
C06023=1076.739,205.409,421.701,174.338,25.610,154.463
C06024=1076.734,205.160,421.726,174.336,25.607,154.462
C06025=1076.728,204.912,421.750,174.334,25.604,154.462
C06026=1076.722,204.664,421.774,174.331,25.602,154.462
C06027=1076.717,204.414,421.798,174.329,25.599,154.462
C06028=1076.711,204.165,421.822,174.326,25.596,154.461
C06029=1076.705,203.917,421.845,174.324,25.594,154.461
C06030=1076.700,203.668,421.870,174.322,25.591,154.461
C06031=1076.695,203.419,421.893,174.319,25.588,154.460
C06032=1076.688,203.170,421.917,174.317,25.586,154.460
C06033=1076.683,202.921,421.942,174.315,25.583,154.460
C06034=1076.678,202.673,421.966,174.312,25.580,154.459
C06035=1076.672,202.424,421.989,174.310,25.577,154.459
C06036=1076.667,202.175,422.013,174.308,25.575,154.459
C06037=1076.660,201.926,422.037,174.306,25.572,154.459
C06038=1076.654,201.677,422.060,174.304,25.570,154.458
C06039=1076.649,201.429,422.084,174.301,25.567,154.458
C06040=1076.643,201.180,422.107,174.299,25.565,154.458
C06041=1076.637,200.931,422.132,174.297,25.562,154.457
C06042=1076.631,200.682,422.155,174.294,25.559,154.457
C06043=1076.626,200.433,422.179,174.292,25.556,154.457
C06044=1076.620,200.185,422.203,174.290,25.554,154.457
C06045=1076.615,199.936,422.226,174.287,25.551,154.456
C06046=1076.609,199.687,422.250,174.285,25.549,154.456
C06047=1076.603,199.438,422.273,174.283,25.546,154.456
C06048=1076.598,199.189,422.297,174.281,25.544,154.455
C06049=1076.592,198.941,422.321,174.279,25.541,154.455
C06050=1076.586,198.692,422.344,174.276,25.538,154.455
C06051=1076.580,198.443,422.369,174.274,25.536,154.455
C06052=1076.574,198.194,422.392,174.271,25.533,154.454
C06053=1076.569,197.945,422.415,174.269,25.531,154.454
C06054=1076.563,197.696,422.439,174.267,25.528,154.454
C06055=1076.558,197.448,422.462,174.264,25.525,154.454
C06056=1076.552,197.199,422.486,174.263,25.523,154.453
C06057=1076.547,196.950,422.509,174.261,25.520,154.453
C06058=1076.540,196.702,422.533,174.258,25.517,154.453
C06059=1076.535,196.452,422.557,174.256,25.515,154.452
C06060=1076.529,196.204,422.580,174.253,25.512,154.452
C06061=1076.523,195.955,422.603,174.251,25.510,154.452
C06062=1076.518,195.705,422.627,174.249,25.507,154.452
C06063=1076.512,195.457,422.650,174.246,25.504,154.451
C06064=1076.506,195.208,422.673,174.245,25.502,154.451
C06065=1076.501,194.959,422.697,174.243,25.499,154.451
C06066=1076.495,194.711,422.720,174.240,25.496,154.450
C06067=1076.490,194.462,422.743,174.238,25.494,154.450
C06068=1076.485,194.213,422.767,174.236,25.491,154.450
C06069=1076.479,193.964,422.791,174.233,25.488,154.450
C06070=1076.473,193.716,422.814,174.232,25.486,154.449
C06071=1076.468,193.466,422.837,174.229,25.484,154.449
C06072=1076.462,193.217,422.860,174.227,25.481,154.449
C06073=1076.456,192.969,422.884,174.225,25.478,154.449
C06074=1076.450,192.719,422.908,174.222,25.476,154.448
C06075=1076.445,192.470,422.931,174.220,25.473,154.448
C06076=1076.439,192.221,422.954,174.218,25.470,154.448
C06077=1076.433,191.973,422.977,174.216,25.468,154.447
C06078=1076.427,191.692,423.003,174.213,25.465,154.447
C06079=1076.421,191.412,423.030,174.211,25.462,154.447
C06080=1076.415,191.131,423.055,174.208,25.459,154.446
C06081=1076.409,190.850,423.082,174.206,25.456,154.446
C06082=1076.403,190.602,423.105,174.204,25.453,154.446
C06083=1076.397,190.353,423.128,174.201,25.451,154.445
C06084=1076.391,190.104,423.152,174.199,25.448,154.445
C06085=1076.386,189.855,423.175,174.197,25.446,154.445
C06086=1076.381,189.606,423.198,174.195,25.443,154.445
C06087=1076.375,189.357,423.221,174.193,25.440,154.444
C06088=1076.369,189.109,423.244,174.190,25.437,154.444
C06089=1076.365,188.860,423.267,174.188,25.435,154.444
C06090=1076.359,188.611,423.290,174.187,25.432,154.443
C06091=1076.353,188.362,423.313,174.184,25.430,154.443
C06092=1076.348,188.113,423.336,174.182,25.427,154.443
C06093=1076.343,187.864,423.360,174.180,25.424,154.443
C06094=1076.337,187.615,423.383,174.177,25.421,154.442
C06095=1076.331,187.366,423.405,174.176,25.419,154.442
C06096=1076.325,187.117,423.428,174.173,25.416,154.442
C06097=1076.320,186.869,423.451,174.171,25.414,154.441
C06098=1076.315,186.620,423.475,174.169,25.411,154.441
C06099=1076.310,186.371,423.497,174.167,25.408,154.441
C06100=1076.304,186.122,423.520,174.165,25.406,154.441
C06101=1076.298,185.873,423.543,174.163,25.403,154.440
C06102=1076.292,185.624,423.566,174.160,25.401,154.440
C06103=1076.287,185.375,423.590,174.158,25.398,154.440
C06104=1076.282,185.126,423.613,174.156,25.396,154.439
C06105=1076.276,184.878,423.635,174.154,25.393,154.439
C06106=1076.271,184.629,423.658,174.152,25.390,154.439
C06107=1076.265,184.380,423.681,174.149,25.388,154.439
C06108=1076.260,184.131,423.703,174.148,25.386,154.438
C06109=1076.253,183.882,423.726,174.146,25.383,154.438
C06110=1076.247,183.633,423.749,174.143,25.380,154.438
C06111=1076.242,183.384,423.772,174.141,25.378,154.438
C06112=1076.236,183.136,423.795,174.139,25.375,154.437
C06113=1076.230,182.887,423.818,174.137,25.373,154.437
C06114=1076.224,182.637,423.839,174.135,25.370,154.437
C06115=1076.218,182.389,423.862,174.132,25.367,154.436
C06116=1076.213,182.140,423.885,174.131,25.365,154.436
C06117=1076.207,181.891,423.908,174.128,25.363,154.436
C06118=1076.200,181.642,423.930,174.126,25.360,154.436
C06119=1076.195,181.393,423.953,174.124,25.358,154.436
C06120=1076.189,181.144,423.976,174.122,25.356,154.435
C06121=1076.184,180.896,423.998,174.120,25.353,154.435
C06122=1076.178,180.646,424.020,174.117,25.350,154.435
C06123=1076.172,180.397,424.043,174.115,25.348,154.434
C06124=1076.166,180.149,424.066,174.114,25.345,154.434
C06125=1076.161,179.900,424.089,174.111,25.343,154.434
C06126=1076.155,179.650,424.110,174.109,25.340,154.434
C06127=1076.149,179.402,424.133,174.107,25.338,154.433
C06128=1076.144,179.153,424.156,174.105,25.335,154.433
C06129=1076.138,178.904,424.178,174.103,25.333,154.433
C06130=1076.132,178.655,424.200,174.100,25.330,154.433
C06131=1076.126,178.406,424.223,174.098,25.327,154.432
C06132=1076.121,178.157,424.246,174.097,25.325,154.432
C06133=1076.115,177.908,424.269,174.094,25.322,154.432
C06134=1076.109,177.659,424.290,174.092,25.320,154.431
C06135=1076.104,177.411,424.313,174.090,25.318,154.431
C06136=1076.098,177.161,424.335,174.088,25.315,154.431
C06137=1076.092,176.912,424.357,174.086,25.312,154.431
C06138=1076.086,176.664,424.380,174.083,25.310,154.430
C06139=1076.081,176.415,424.402,174.082,25.307,154.430
C06140=1076.075,176.166,424.425,174.080,25.305,154.430
C06141=1076.069,175.917,424.447,174.077,25.302,154.430
C06142=1076.063,175.636,424.472,174.075,25.299,154.429
C06143=1076.057,175.355,424.497,174.073,25.296,154.429
C06144=1076.050,175.074,424.522,174.070,25.294,154.429
C06145=1076.044,174.793,424.548,174.068,25.291,154.428
C06146=1076.038,174.544,424.570,174.066,25.288,154.428
C06147=1076.032,174.295,424.592,174.064,25.286,154.428
C06148=1076.027,174.046,424.614,174.062,25.283,154.428
C06149=1076.021,173.797,424.637,174.059,25.281,154.427
C06150=1076.015,173.548,424.659,174.058,25.279,154.427
C06151=1076.010,173.299,424.681,174.056,25.275,154.427
C06152=1076.005,173.050,424.704,174.053,25.273,154.426
C06153=1075.999,172.801,424.725,174.052,25.270,154.426
C06154=1075.993,172.553,424.748,174.050,25.268,154.426
C06155=1075.988,172.303,424.770,174.047,25.265,154.426
C06156=1075.982,172.054,424.792,174.046,25.263,154.425
C06157=1075.976,171.805,424.815,174.043,25.260,154.425
C06158=1075.971,171.556,424.836,174.041,25.258,154.425
C06159=1075.965,171.307,424.858,174.040,25.255,154.424
C06160=1075.960,171.059,424.881,174.037,25.253,154.424
C06161=1075.954,170.810,424.902,174.035,25.250,154.424
C06162=1075.948,170.560,424.924,174.034,25.248,154.424
C06163=1075.943,170.312,424.947,174.031,25.245,154.423
C06164=1075.937,170.063,424.969,174.029,25.243,154.423
C06165=1075.932,169.813,424.991,174.027,25.240,154.423
C06166=1075.927,169.565,425.013,174.025,25.238,154.423
C06167=1075.920,169.316,425.035,174.023,25.235,154.422
C06168=1075.915,169.067,425.057,174.021,25.233,154.422
C06169=1075.909,168.818,425.079,174.019,25.229,154.422
C06170=1075.904,168.568,425.101,174.017,25.227,154.421
C06171=1075.898,168.321,425.123,174.015,25.225,154.421
C06172=1075.893,168.071,425.145,174.013,25.222,154.421
C06173=1075.888,167.822,425.167,174.011,25.220,154.420
C06174=1075.882,167.573,425.189,174.009,25.217,154.420
C06175=1075.876,167.324,425.211,174.007,25.214,154.420
C06176=1075.871,167.075,425.232,174.005,25.212,154.420
C06177=1075.865,166.826,425.255,174.003,25.209,154.419
C06178=1075.859,166.578,425.276,174.001,25.207,154.419
C06179=1075.854,166.328,425.299,173.999,25.204,154.419
C06180=1075.849,166.079,425.320,173.997,25.201,154.418
C06181=1075.843,165.830,425.342,173.996,25.199,154.418
C06182=1075.838,165.581,425.364,173.993,25.196,154.418
C06183=1075.832,165.332,425.386,173.991,25.194,154.418
C06184=1075.827,165.083,425.407,173.989,25.191,154.417
C06185=1075.821,164.834,425.429,173.987,25.189,154.417
C06186=1075.816,164.586,425.452,173.985,25.186,154.417
C06187=1075.810,164.337,425.473,173.983,25.183,154.416
C06188=1075.805,164.088,425.495,173.981,25.181,154.416
C06189=1075.799,163.839,425.517,173.980,25.178,154.416
C06190=1075.794,163.590,425.539,173.977,25.176,154.416
C06191=1075.788,163.341,425.560,173.975,25.173,154.415
C06192=1075.783,163.092,425.582,173.973,25.171,154.415
C06193=1075.777,162.843,425.604,173.971,25.168,154.415
C06194=1075.772,162.594,425.626,173.970,25.165,154.414
C06195=1075.766,162.345,425.647,173.968,25.163,154.414
C06196=1075.761,162.096,425.669,173.965,25.160,154.414
C06197=1075.755,161.847,425.691,173.964,25.158,154.414
C06198=1075.750,161.598,425.713,173.961,25.155,154.413
C06199=1075.744,161.348,425.734,173.960,25.153,154.413
C06200=1075.739,161.099,425.755,173.958,25.150,154.413
C06201=1075.733,160.850,425.777,173.955,25.147,154.412
C06202=1075.728,160.601,425.798,173.954,25.145,154.412
C06203=1075.721,160.352,425.820,173.951,25.143,154.412
C06204=1075.717,160.103,425.842,173.950,25.140,154.412
C06205=1075.710,159.854,425.863,173.948,25.138,154.411
C06206=1075.704,159.573,425.888,173.946,25.134,154.411
C06207=1075.698,159.291,425.912,173.943,25.132,154.411
C06208=1075.691,159.010,425.936,173.941,25.129,154.410
C06209=1075.685,158.729,425.960,173.939,25.126,154.410
C06210=1075.679,158.480,425.982,173.937,25.124,154.410
C06211=1075.674,158.231,426.002,173.935,25.121,154.410
C06212=1075.668,157.982,426.024,173.933,25.119,154.409
C06213=1075.663,157.733,426.046,173.931,25.116,154.409
C06214=1075.657,157.484,426.067,173.930,25.114,154.409
C06215=1075.651,157.235,426.089,173.927,25.111,154.408
C06216=1075.645,156.985,426.109,173.925,25.108,154.408
C06217=1075.640,156.737,426.131,173.924,25.106,154.408
C06218=1075.634,156.488,426.152,173.921,25.103,154.408
C06219=1075.629,156.238,426.174,173.920,25.101,154.407
C06220=1075.623,155.990,426.195,173.918,25.098,154.407
C06221=1075.617,155.741,426.216,173.916,25.096,154.407
C06222=1075.612,155.492,426.238,173.914,25.093,154.406
C06223=1075.606,155.242,426.259,173.912,25.091,154.406
C06224=1075.600,154.994,426.280,173.910,25.088,154.406
C06225=1075.594,154.745,426.302,173.908,25.085,154.406
C06226=1075.589,154.495,426.322,173.906,25.083,154.405
C06227=1075.583,154.247,426.343,173.904,25.080,154.405
C06228=1075.577,153.998,426.365,173.903,25.078,154.405
C06229=1075.572,153.749,426.386,173.900,25.075,154.404
C06230=1075.566,153.499,426.407,173.899,25.073,154.404
C06231=1075.561,153.250,426.428,173.896,25.071,154.404
C06232=1075.555,153.002,426.449,173.895,25.068,154.404
C06233=1075.549,152.753,426.471,173.893,25.066,154.403
C06234=1075.544,152.503,426.491,173.891,25.063,154.403
C06235=1075.537,152.254,426.513,173.889,25.061,154.403
C06236=1075.533,152.005,426.534,173.887,25.058,154.403
C06237=1075.527,151.756,426.555,173.885,25.056,154.402
C06238=1075.521,151.507,426.576,173.883,25.053,154.402
C06239=1075.516,151.258,426.597,173.881,25.051,154.402
C06240=1075.511,151.009,426.618,173.879,25.048,154.401
C06241=1075.504,150.760,426.639,173.878,25.046,154.401
C06242=1075.498,150.511,426.660,173.875,25.043,154.401
C06243=1075.493,150.262,426.681,173.874,25.040,154.401
C06244=1075.487,150.013,426.702,173.872,25.038,154.400
C06245=1075.481,149.764,426.723,173.870,25.035,154.400
C06246=1075.476,149.515,426.744,173.868,25.033,154.400
C06247=1075.470,149.266,426.765,173.866,25.030,154.399
C06248=1075.465,149.017,426.786,173.864,25.028,154.399
C06249=1075.459,148.768,426.807,173.863,25.025,154.399
C06250=1075.453,148.518,426.828,173.860,25.023,154.399
C06251=1075.448,148.269,426.849,173.859,25.020,154.398
C06252=1075.443,148.021,426.870,173.857,25.018,154.398
C06253=1075.437,147.771,426.891,173.855,25.015,154.398
C06254=1075.430,147.523,426.911,173.853,25.013,154.398
C06255=1075.425,147.273,426.932,173.851,25.010,154.397
C06256=1075.419,147.024,426.953,173.849,25.008,154.397
C06257=1075.414,146.775,426.974,173.848,25.005,154.397
C06258=1075.408,146.526,426.995,173.845,25.003,154.396
C06259=1075.402,146.277,427.015,173.844,25.000,154.396
C06260=1075.396,146.028,427.036,173.842,24.998,154.396
C06261=1075.391,145.779,427.057,173.840,24.995,154.396
C06262=1075.385,145.529,427.078,173.838,24.993,154.395
C06263=1075.379,145.281,427.098,173.836,24.991,154.395
C06264=1075.374,145.032,427.119,173.834,24.987,154.395
C06265=1075.368,144.783,427.140,173.833,24.985,154.394
C06266=1075.363,144.533,427.160,173.831,24.982,154.394
C06267=1075.357,144.284,427.182,173.829,24.980,154.394
C06268=1075.351,144.035,427.202,173.827,24.977,154.394
C06269=1075.346,143.786,427.222,173.825,24.975,154.393
C06270=1075.339,143.505,427.246,173.823,24.972,154.393
C06271=1075.333,143.223,427.269,173.821,24.969,154.393
C06272=1075.326,142.941,427.292,173.819,24.967,154.392
C06273=1075.319,142.660,427.316,173.817,24.964,154.392
C06274=1075.314,142.410,427.336,173.815,24.961,154.392
C06275=1075.309,142.161,427.357,173.814,24.959,154.391
C06276=1075.304,141.912,427.377,173.811,24.956,154.391
C06277=1075.297,141.663,427.398,173.810,24.954,154.391
C06278=1075.292,141.414,427.419,173.807,24.951,154.391
C06279=1075.286,141.165,427.440,173.806,24.949,154.390
C06280=1075.280,140.916,427.460,173.804,24.946,154.390
C06281=1075.275,140.667,427.480,173.802,24.943,154.390
C06282=1075.270,140.418,427.501,173.800,24.941,154.389
C06283=1075.263,140.169,427.521,173.799,24.938,154.389
C06284=1075.258,139.919,427.542,173.796,24.936,154.389
C06285=1075.253,139.670,427.562,173.795,24.933,154.389
C06286=1075.246,139.422,427.583,173.793,24.931,154.388
C06287=1075.241,139.172,427.604,173.791,24.928,154.388
C06288=1075.235,138.923,427.624,173.790,24.926,154.388
C06289=1075.229,138.674,427.644,173.787,24.923,154.387
C06290=1075.224,138.425,427.665,173.786,24.921,154.387
C06291=1075.218,138.176,427.685,173.784,24.918,154.387
C06292=1075.213,137.927,427.705,173.782,24.916,154.387
C06293=1075.206,137.678,427.726,173.780,24.913,154.386
C06294=1075.201,137.429,427.746,173.779,24.910,154.386
C06295=1075.195,137.180,427.766,173.776,24.908,154.386
C06296=1075.190,136.931,427.787,173.775,24.905,154.385
C06297=1075.184,136.682,427.807,173.774,24.903,154.385
C06298=1075.178,136.433,427.827,173.771,24.900,154.385
C06299=1075.172,136.183,427.847,173.770,24.898,154.385
C06300=1075.167,135.934,427.868,173.768,24.895,154.384
C06301=1075.161,135.685,427.887,173.766,24.893,154.384
C06302=1075.156,135.436,427.908,173.764,24.890,154.384
C06303=1075.150,135.187,427.928,173.762,24.888,154.383
C06304=1075.144,134.938,427.948,173.760,24.885,154.383
C06305=1075.138,134.689,427.968,173.759,24.883,154.383
C06306=1075.133,134.440,427.989,173.757,24.880,154.382
C06307=1075.127,134.190,428.009,173.755,24.878,154.382
C06308=1075.121,133.941,428.030,173.754,24.875,154.382
C06309=1075.115,133.692,428.050,173.751,24.873,154.382
C06310=1075.110,133.442,428.070,173.750,24.870,154.381
C06311=1075.104,133.194,428.090,173.748,24.868,154.381
C06312=1075.099,132.945,428.110,173.746,24.865,154.381
C06313=1075.093,132.696,428.130,173.745,24.862,154.380
C06314=1075.088,132.447,428.151,173.743,24.860,154.380
C06315=1075.082,132.197,428.170,173.741,24.857,154.380
C06316=1075.077,131.948,428.190,173.739,24.855,154.380
C06317=1075.070,131.699,428.211,173.737,24.852,154.379
C06318=1075.064,131.450,428.231,173.736,24.850,154.379
C06319=1075.058,131.201,428.251,173.734,24.847,154.379
C06320=1075.053,130.951,428.270,173.732,24.845,154.378
C06321=1075.047,130.702,428.290,173.730,24.842,154.378
C06322=1075.041,130.454,428.310,173.729,24.840,154.378
C06323=1075.036,130.204,428.330,173.726,24.837,154.378
C06324=1075.030,129.955,428.350,173.725,24.835,154.377
C06325=1075.024,129.706,428.370,173.723,24.833,154.377
C06326=1075.018,129.457,428.390,173.721,24.830,154.377
C06327=1075.012,129.207,428.410,173.720,24.828,154.377
C06328=1075.006,128.958,428.430,173.717,24.825,154.376
C06329=1075.001,128.709,428.450,173.716,24.823,154.376
C06330=1074.995,128.460,428.469,173.715,24.820,154.376
C06331=1074.989,128.211,428.489,173.712,24.817,154.375
C06332=1074.983,127.962,428.509,173.711,24.815,154.375
C06333=1074.978,127.713,428.529,173.709,24.812,154.375
C06334=1074.971,127.430,428.551,173.707,24.810,154.374
C06335=1074.965,127.150,428.574,173.705,24.807,154.374
C06336=1074.958,126.868,428.596,173.703,24.804,154.374
C06337=1074.951,126.586,428.618,173.702,24.801,154.373
C06338=1074.945,126.337,428.638,173.699,24.799,154.373
C06339=1074.940,126.087,428.658,173.698,24.796,154.373
C06340=1074.934,125.838,428.678,173.696,24.794,154.373
C06341=1074.929,125.589,428.697,173.694,24.791,154.372
C06342=1074.923,125.340,428.717,173.693,24.789,154.372
C06343=1074.917,125.091,428.737,173.690,24.786,154.372
C06344=1074.911,124.842,428.757,173.689,24.783,154.371
C06345=1074.906,124.593,428.777,173.688,24.781,154.371
C06346=1074.900,124.343,428.796,173.685,24.778,154.371
C06347=1074.894,124.094,428.816,173.684,24.776,154.371
C06348=1074.888,123.845,428.836,173.682,24.773,154.370
C06349=1074.883,123.597,428.855,173.680,24.771,154.370
C06350=1074.877,123.347,428.874,173.679,24.769,154.370
C06351=1074.872,123.098,428.894,173.677,24.765,154.369
C06352=1074.866,122.849,428.914,173.675,24.763,154.369
C06353=1074.861,122.599,428.933,173.674,24.761,154.369
C06354=1074.855,122.351,428.953,173.672,24.758,154.369
C06355=1074.849,122.101,428.973,173.670,24.756,154.368
C06356=1074.843,121.852,428.993,173.668,24.753,154.368
C06357=1074.837,121.603,429.012,173.667,24.750,154.368
C06358=1074.832,121.353,429.032,173.665,24.748,154.367
C06359=1074.826,121.104,429.052,173.663,24.745,154.367
C06360=1074.821,120.855,429.071,173.662,24.743,154.367
C06361=1074.815,120.606,429.091,173.660,24.741,154.366
C06362=1074.809,120.357,429.110,173.658,24.738,154.366
C06363=1074.804,120.108,429.129,173.657,24.735,154.366
C06364=1074.798,119.859,429.149,173.655,24.733,154.365
C06365=1074.792,119.610,429.168,173.653,24.730,154.365
C06366=1074.787,119.360,429.187,173.652,24.728,154.365
C06367=1074.781,119.111,429.207,173.650,24.725,154.365
C06368=1074.776,118.862,429.227,173.648,24.722,154.364
C06369=1074.770,118.612,429.247,173.647,24.720,154.364
C06370=1074.764,118.363,429.266,173.644,24.717,154.364
C06371=1074.759,118.115,429.285,173.643,24.715,154.363
C06372=1074.753,117.865,429.305,173.642,24.712,154.363
C06373=1074.747,117.616,429.324,173.639,24.709,154.363
C06374=1074.741,117.367,429.344,173.638,24.707,154.362
C06375=1074.736,117.118,429.363,173.637,24.704,154.362
C06376=1074.730,116.868,429.382,173.634,24.701,154.362
C06377=1074.725,116.619,429.401,173.633,24.699,154.362
C06378=1074.719,116.371,429.421,173.632,24.697,154.361
C06379=1074.713,116.121,429.440,173.629,24.694,154.361
C06380=1074.708,115.872,429.460,173.628,24.691,154.361
C06381=1074.702,115.622,429.479,173.627,24.689,154.360
C06382=1074.698,115.373,429.498,173.624,24.686,154.360
C06383=1074.692,115.124,429.518,173.623,24.683,154.360
C06384=1074.686,114.875,429.538,173.622,24.681,154.359
C06385=1074.680,114.626,429.557,173.619,24.678,154.359
C06386=1074.675,114.376,429.576,173.618,24.676,154.359
C06387=1074.669,114.127,429.595,173.617,24.673,154.358
C06388=1074.663,113.878,429.614,173.614,24.670,154.358
C06389=1074.657,113.629,429.633,173.613,24.668,154.358
C06390=1074.651,113.380,429.653,173.612,24.666,154.358
C06391=1074.646,113.131,429.672,173.609,24.663,154.357
C06392=1074.640,112.881,429.691,173.608,24.660,154.357
C06393=1074.635,112.632,429.710,173.607,24.658,154.357
C06394=1074.629,112.383,429.729,173.604,24.655,154.356
C06395=1074.623,112.134,429.748,173.603,24.653,154.356
C06396=1074.617,111.884,429.767,173.602,24.650,154.356
C06397=1074.611,111.635,429.786,173.599,24.647,154.355
C06398=1074.605,111.354,429.808,173.598,24.645,154.355
C06399=1074.599,111.072,429.829,173.596,24.641,154.355
C06400=1074.592,110.790,429.851,173.595,24.639,154.354
C06401=1074.586,110.509,429.873,173.592,24.636,154.354
C06402=1074.579,110.259,429.892,173.591,24.634,154.354
C06403=1074.573,110.010,429.911,173.589,24.631,154.353
C06404=1074.569,109.761,429.929,173.587,24.628,154.353
C06405=1074.563,109.511,429.948,173.586,24.626,154.353
C06406=1074.557,109.262,429.967,173.584,24.623,154.353
C06407=1074.551,109.013,429.986,173.582,24.621,154.352
C06408=1074.545,108.763,430.005,173.581,24.618,154.352
C06409=1074.539,108.515,430.024,173.580,24.616,154.352
C06410=1074.534,108.265,430.043,173.577,24.613,154.351
C06411=1074.528,108.016,430.062,173.576,24.610,154.351
C06412=1074.522,107.767,430.081,173.575,24.608,154.351
C06413=1074.516,107.518,430.100,173.572,24.605,154.350
C06414=1074.511,107.269,430.119,173.571,24.603,154.350
C06415=1074.504,107.019,430.138,173.570,24.600,154.350
C06416=1074.499,106.770,430.157,173.567,24.597,154.349
C06417=1074.494,106.521,430.175,173.566,24.595,154.349
C06418=1074.487,106.272,430.194,173.565,24.593,154.349
C06419=1074.482,106.022,430.213,173.563,24.589,154.349
C06420=1074.477,105.773,430.232,173.561,24.587,154.348
C06421=1074.470,105.524,430.250,173.560,24.585,154.348
C06422=1074.465,105.275,430.270,173.558,24.582,154.348
C06423=1074.459,105.025,430.288,173.556,24.579,154.347
C06424=1074.453,104.776,430.306,173.555,24.577,154.347
C06425=1074.448,104.527,430.326,173.553,24.574,154.347
C06426=1074.442,104.278,430.345,173.551,24.572,154.346
C06427=1074.436,104.029,430.363,173.550,24.569,154.346
C06428=1074.431,103.779,430.382,173.549,24.567,154.346
C06429=1074.425,103.530,430.401,173.547,24.564,154.345
C06430=1074.419,103.281,430.419,173.545,24.561,154.345
C06431=1074.414,103.032,430.439,173.544,24.559,154.345
C06432=1074.407,102.782,430.456,173.542,24.556,154.344
C06433=1074.402,102.533,430.475,173.540,24.554,154.344
C06434=1074.397,102.284,430.495,173.539,24.551,154.344
C06435=1074.390,102.035,430.513,173.537,24.548,154.344
C06436=1074.385,101.785,430.531,173.536,24.546,154.343
C06437=1074.380,101.536,430.551,173.534,24.543,154.343
C06438=1074.374,101.288,430.569,173.532,24.540,154.343
C06439=1074.369,101.037,430.587,173.531,24.538,154.342
C06440=1074.362,100.788,430.606,173.529,24.535,154.342
C06441=1074.356,100.539,430.625,173.527,24.533,154.342
C06442=1074.351,100.290,430.643,173.526,24.530,154.341
C06443=1074.344,100.041,430.662,173.525,24.528,154.341
C06444=1074.339,99.791,430.681,173.522,24.525,154.341
C06445=1074.333,99.542,430.698,173.521,24.523,154.341
C06446=1074.328,99.293,430.718,173.520,24.520,154.340
C06447=1074.321,99.043,430.736,173.518,24.517,154.340
C06448=1074.316,98.795,430.754,173.516,24.515,154.340
C06449=1074.310,98.545,430.773,173.515,24.512,154.339
C06450=1074.304,98.296,430.791,173.513,24.510,154.339
C06451=1074.299,98.047,430.810,173.511,24.507,154.339
C06452=1074.293,97.797,430.828,173.510,24.504,154.338
C06453=1074.287,97.549,430.846,173.508,24.502,154.338
C06454=1074.281,97.299,430.865,173.507,24.500,154.338
C06455=1074.275,97.049,430.883,173.505,24.497,154.337
C06456=1074.270,96.801,430.902,173.504,24.494,154.337
C06457=1074.264,96.551,430.920,173.502,24.492,154.337
C06458=1074.258,96.303,430.938,173.501,24.489,154.336
C06459=1074.253,96.053,430.957,173.499,24.486,154.336
C06460=1074.246,95.803,430.976,173.497,24.484,154.336
C06461=1074.241,95.554,430.993,173.496,24.482,154.336
C06462=1074.235,95.272,431.014,173.494,24.478,154.335
C06463=1074.228,94.991,431.035,173.493,24.475,154.335
C06464=1074.222,94.709,431.056,173.490,24.473,154.335
C06465=1074.215,94.427,431.076,173.489,24.470,154.334
C06466=1074.209,94.178,431.095,173.487,24.467,154.334
C06467=1074.204,93.929,431.113,173.486,24.464,154.333
C06468=1074.197,93.680,431.131,173.484,24.462,154.333
C06469=1074.192,93.430,431.150,173.483,24.459,154.333
C06470=1074.186,93.181,431.167,173.481,24.456,154.332
C06471=1074.180,92.932,431.186,173.479,24.454,154.332
C06472=1074.175,92.682,431.204,173.478,24.452,154.332
C06473=1074.169,92.434,431.223,173.477,24.449,154.331
C06474=1074.163,92.184,431.240,173.474,24.446,154.331
C06475=1074.158,91.935,431.259,173.473,24.444,154.331
C06476=1074.152,91.686,431.277,173.472,24.441,154.331
C06477=1074.146,91.437,431.295,173.470,24.438,154.330
C06478=1074.141,91.186,431.313,173.468,24.436,154.330
C06479=1074.135,90.938,431.332,173.467,24.433,154.330
C06480=1074.129,90.688,431.350,173.466,24.430,154.329
C06481=1074.124,90.439,431.367,173.464,24.428,154.329
C06482=1074.117,90.190,431.386,173.462,24.425,154.329
C06483=1074.112,89.940,431.404,173.461,24.422,154.328
C06484=1074.106,89.691,431.422,173.459,24.420,154.328
C06485=1074.100,89.441,431.440,173.458,24.418,154.328
C06486=1074.094,89.193,431.458,173.457,24.415,154.327
C06487=1074.088,88.943,431.476,173.454,24.412,154.327
C06488=1074.083,88.694,431.494,173.453,24.410,154.327
C06489=1074.077,88.444,431.512,173.452,24.407,154.327
C06490=1074.071,88.196,431.530,173.450,24.405,154.326
C06491=1074.065,87.946,431.548,173.448,24.402,154.326
C06492=1074.060,87.697,431.566,173.447,24.399,154.326
C06493=1074.054,87.447,431.584,173.445,24.397,154.325
C06494=1074.048,87.198,431.601,173.444,24.395,154.325
C06495=1074.042,86.949,431.620,173.442,24.391,154.325
C06496=1074.036,86.700,431.638,173.441,24.389,154.324
C06497=1074.030,86.450,431.656,173.439,24.387,154.324
C06498=1074.025,86.201,431.673,173.438,24.384,154.324
C06499=1074.018,85.951,431.691,173.436,24.381,154.323
C06500=1074.013,85.703,431.709,173.434,24.379,154.323
C06501=1074.007,85.454,431.727,173.433,24.376,154.323
C06502=1074.001,85.204,431.745,173.432,24.373,154.322
C06503=1073.995,84.955,431.762,173.430,24.371,154.322
C06504=1073.989,84.705,431.780,173.428,24.368,154.322
C06505=1073.985,84.456,431.799,173.427,24.366,154.321
C06506=1073.978,84.206,431.816,173.425,24.363,154.321
C06507=1073.973,83.957,431.834,173.424,24.361,154.321
C06508=1073.967,83.708,431.852,173.422,24.358,154.321
C06509=1073.961,83.458,431.870,173.421,24.355,154.320
C06510=1073.955,83.210,431.888,173.419,24.353,154.320
C06511=1073.949,82.960,431.906,173.418,24.350,154.320
C06512=1073.944,82.711,431.923,173.417,24.348,154.319
C06513=1073.938,82.462,431.941,173.414,24.345,154.319
C06514=1073.932,82.212,431.959,173.413,24.342,154.319
C06515=1073.927,81.963,431.976,173.412,24.340,154.318
C06516=1073.921,81.714,431.994,173.410,24.337,154.318
C06517=1073.915,81.465,432.012,173.409,24.334,154.318
C06518=1073.910,81.216,432.029,173.407,24.332,154.317
C06519=1073.903,80.966,432.047,173.406,24.329,154.317
C06520=1073.898,80.717,432.065,173.404,24.326,154.317
C06521=1073.892,80.467,432.083,173.403,24.324,154.316
C06522=1073.886,80.218,432.100,173.401,24.321,154.316
C06523=1073.881,79.969,432.118,173.399,24.318,154.316
C06524=1073.875,79.719,432.136,173.398,24.316,154.315
C06525=1073.869,79.470,432.154,173.397,24.313,154.315
C06526=1073.863,79.188,432.173,173.395,24.310,154.315
C06527=1073.856,78.907,432.193,173.393,24.307,154.314
C06528=1073.850,78.625,432.213,173.391,24.304,154.314
C06529=1073.843,78.343,432.233,173.390,24.301,154.314
C06530=1073.838,78.094,432.250,173.389,24.299,154.313
C06531=1073.832,77.845,432.268,173.387,24.296,154.313
C06532=1073.825,77.595,432.285,173.385,24.293,154.313
C06533=1073.820,77.346,432.303,173.384,24.291,154.312
C06534=1073.814,77.097,432.320,173.382,24.289,154.312
C06535=1073.808,76.847,432.338,173.381,24.286,154.312
C06536=1073.803,76.598,432.356,173.379,24.283,154.311
C06537=1073.798,76.349,432.373,173.378,24.281,154.311
C06538=1073.791,76.099,432.390,173.376,24.278,154.311
C06539=1073.785,75.850,432.407,173.375,24.275,154.310
C06540=1073.780,75.601,432.425,173.374,24.273,154.310
C06541=1073.773,75.351,432.443,173.372,24.270,154.310
C06542=1073.768,75.102,432.459,173.370,24.267,154.309
C06543=1073.762,74.853,432.477,173.369,24.265,154.309
C06544=1073.756,74.603,432.495,173.368,24.262,154.309
C06545=1073.750,74.354,432.512,173.366,24.260,154.308
C06546=1073.745,74.105,432.530,173.364,24.257,154.308
C06547=1073.738,73.855,432.546,173.363,24.254,154.308
C06548=1073.733,73.606,432.564,173.361,24.252,154.307
C06549=1073.727,73.357,432.582,173.360,24.249,154.307
C06550=1073.722,73.107,432.598,173.359,24.246,154.307
C06551=1073.715,72.858,432.616,173.357,24.244,154.307
C06552=1073.710,72.609,432.633,173.355,24.241,154.306
C06553=1073.704,72.360,432.651,173.354,24.238,154.306
C06554=1073.698,72.110,432.668,173.353,24.236,154.306
C06555=1073.692,71.861,432.685,173.351,24.234,154.305
C06556=1073.687,71.612,432.703,173.350,24.231,154.305
C06557=1073.681,71.362,432.720,173.348,24.228,154.305
C06558=1073.674,71.113,432.737,173.347,24.225,154.304
C06559=1073.669,70.864,432.754,173.345,24.223,154.304
C06560=1073.664,70.614,432.771,173.344,24.220,154.304
C06561=1073.658,70.365,432.789,173.343,24.217,154.303
C06562=1073.651,70.116,432.806,173.340,24.215,154.303
C06563=1073.646,69.866,432.823,173.339,24.212,154.303
C06564=1073.641,69.617,432.841,173.338,24.209,154.302
C06565=1073.635,69.367,432.857,173.337,24.207,154.302
C06566=1073.629,69.118,432.875,173.335,24.205,154.302
C06567=1073.622,68.869,432.892,173.333,24.201,154.301
C06568=1073.617,68.619,432.909,173.332,24.199,154.301
C06569=1073.612,68.370,432.926,173.330,24.197,154.301
C06570=1073.606,68.121,432.942,173.329,24.194,154.300
C06571=1073.600,67.871,432.960,173.328,24.191,154.300
C06572=1073.594,67.622,432.977,173.326,24.189,154.300
C06573=1073.588,67.373,432.994,173.324,24.186,154.299
C06574=1073.583,67.123,433.011,173.323,24.183,154.299
C06575=1073.576,66.874,433.028,173.322,24.181,154.299
C06576=1073.570,66.625,433.046,173.320,24.178,154.298
C06577=1073.565,66.375,433.062,173.319,24.176,154.298
C06578=1073.559,66.126,433.080,173.318,24.173,154.298
C06579=1073.553,65.877,433.096,173.316,24.170,154.297
C06580=1073.547,65.627,433.113,173.314,24.168,154.297
C06581=1073.541,65.378,433.130,173.313,24.165,154.297
C06582=1073.536,65.128,433.147,173.312,24.162,154.296
C06583=1073.530,64.879,433.164,173.310,24.160,154.296
C06584=1073.524,64.630,433.181,173.308,24.157,154.296
C06585=1073.517,64.380,433.198,173.307,24.154,154.296
C06586=1073.512,64.131,433.215,173.306,24.152,154.295
C06587=1073.506,63.882,433.232,173.304,24.150,154.295
C06588=1073.500,63.633,433.248,173.303,24.147,154.295
C06589=1073.495,63.383,433.265,173.302,24.144,154.294
C06590=1073.488,63.101,433.284,173.300,24.141,154.294
C06591=1073.480,62.819,433.303,173.298,24.139,154.294
C06592=1073.474,62.538,433.323,173.296,24.135,154.293
C06593=1073.467,62.256,433.342,173.295,24.132,154.293
C06594=1073.461,62.006,433.358,173.294,24.130,154.293
C06595=1073.456,61.757,433.375,173.291,24.127,154.292
C06596=1073.450,61.508,433.392,173.290,24.125,154.292
C06597=1073.444,61.259,433.408,173.289,24.122,154.292
C06598=1073.438,61.008,433.425,173.287,24.120,154.291
C06599=1073.432,60.760,433.442,173.286,24.117,154.291
C06600=1073.426,60.510,433.459,173.285,24.114,154.291
C06601=1073.420,60.261,433.475,173.283,24.112,154.290
C06602=1073.414,60.012,433.492,173.281,24.109,154.290
C06603=1073.408,59.762,433.509,173.280,24.107,154.290
C06604=1073.402,59.512,433.525,173.279,24.104,154.289
C06605=1073.396,59.263,433.543,173.277,24.102,154.289
C06606=1073.390,59.014,433.559,173.276,24.099,154.289
C06607=1073.384,58.765,433.575,173.274,24.096,154.288
C06608=1073.378,58.515,433.592,173.273,24.094,154.288
C06609=1073.373,58.266,433.609,173.271,24.091,154.288
C06610=1073.367,58.017,433.625,173.270,24.088,154.287
C06611=1073.360,57.767,433.642,173.269,24.086,154.287
C06612=1073.355,57.517,433.659,173.267,24.083,154.287
C06613=1073.349,57.268,433.675,173.266,24.081,154.287
C06614=1073.343,57.019,433.692,173.264,24.078,154.286
C06615=1073.337,56.770,433.708,173.262,24.075,154.286
C06616=1073.332,56.520,433.725,173.261,24.073,154.286
C06617=1073.326,56.271,433.742,173.260,24.070,154.285
C06618=1073.320,56.021,433.758,173.259,24.068,154.285
C06619=1073.314,55.773,433.775,173.257,24.065,154.285
C06620=1073.308,55.523,433.792,173.255,24.062,154.284
C06621=1073.302,55.274,433.808,173.254,24.060,154.284
C06622=1073.296,55.024,433.824,173.252,24.057,154.284
C06623=1073.290,54.774,433.841,173.251,24.054,154.283
C06624=1073.285,54.525,433.858,173.250,24.052,154.283
C06625=1073.279,54.275,433.874,173.249,24.050,154.283
C06626=1073.273,54.026,433.890,173.246,24.046,154.282
C06627=1073.267,53.777,433.906,173.245,24.044,154.282
C06628=1073.261,53.528,433.923,173.244,24.041,154.282
C06629=1073.255,53.278,433.940,173.243,24.039,154.281
C06630=1073.249,53.029,433.956,173.241,24.036,154.281
C06631=1073.243,52.780,433.973,173.240,24.033,154.281
C06632=1073.238,52.530,433.989,173.239,24.031,154.280
C06633=1073.232,52.281,434.005,173.236,24.028,154.280
C06634=1073.226,52.031,434.022,173.235,24.025,154.280
C06635=1073.220,51.782,434.038,173.234,24.023,154.279
C06636=1073.214,51.532,434.055,173.233,24.021,154.279
C06637=1073.209,51.283,434.071,173.231,24.018,154.279
C06638=1073.203,51.034,434.087,173.230,24.015,154.278
C06639=1073.197,50.784,434.104,173.229,24.012,154.278
C06640=1073.191,50.535,434.120,173.227,24.010,154.278
C06641=1073.185,50.285,434.136,173.225,24.007,154.278
C06642=1073.180,50.036,434.153,173.224,24.004,154.277
C06643=1073.174,49.787,434.169,173.223,24.002,154.277
C06644=1073.168,49.537,434.186,173.222,23.999,154.276
C06645=1073.162,49.288,434.202,173.220,23.997,154.276
C06646=1073.156,49.038,434.218,173.219,23.994,154.276
C06647=1073.150,48.789,434.235,173.217,23.991,154.275
C06648=1073.145,48.540,434.250,173.215,23.989,154.275
C06649=1073.139,48.291,434.267,173.214,23.986,154.275
C06650=1073.134,48.041,434.283,173.213,23.983,154.274
C06651=1073.128,47.791,434.299,173.212,23.981,154.274
C06652=1073.122,47.542,434.315,173.210,23.978,154.274
C06653=1073.116,47.293,434.332,173.209,23.975,154.274
C06654=1073.110,47.011,434.350,173.207,23.972,154.273
C06655=1073.103,46.728,434.368,173.206,23.969,154.273
C06656=1073.096,46.447,434.387,173.204,23.966,154.272
C06657=1073.090,46.164,434.406,173.203,23.963,154.272
C06658=1073.085,45.916,434.422,173.201,23.961,154.272
C06659=1073.079,45.666,434.437,173.200,23.958,154.271
C06660=1073.073,45.416,434.453,173.198,23.955,154.271
C06661=1073.067,45.167,434.470,173.196,23.953,154.271
C06662=1073.061,44.918,434.486,173.195,23.950,154.270
C06663=1073.055,44.668,434.502,173.194,23.947,154.270
C06664=1073.050,44.418,434.518,173.193,23.944,154.270
C06665=1073.045,44.169,434.534,173.191,23.942,154.269
C06666=1073.039,43.920,434.550,173.190,23.940,154.269
C06667=1073.033,43.671,434.567,173.189,23.937,154.269
C06668=1073.027,43.421,434.583,173.187,23.934,154.268
C06669=1073.022,43.171,434.598,173.185,23.931,154.268
C06670=1073.016,42.922,434.615,173.184,23.929,154.268
C06671=1073.009,42.673,434.630,173.183,23.926,154.267
C06672=1073.003,42.424,434.647,173.181,23.924,154.267
C06673=1072.997,42.174,434.662,173.180,23.921,154.267
C06674=1072.992,41.924,434.678,173.179,23.918,154.266
C06675=1072.986,41.676,434.694,173.177,23.916,154.266
C06676=1072.981,41.426,434.710,173.176,23.913,154.266
C06677=1072.975,41.176,434.726,173.174,23.910,154.265
C06678=1072.969,40.927,434.742,173.173,23.907,154.265
C06679=1072.963,40.677,434.758,173.172,23.905,154.265
C06680=1072.957,40.428,434.774,173.170,23.903,154.265
C06681=1072.951,40.178,434.790,173.169,23.900,154.264
C06682=1072.945,39.929,434.805,173.168,23.897,154.264
C06683=1072.939,39.680,434.821,173.166,23.895,154.264
C06684=1072.933,39.431,434.838,173.164,23.892,154.263
C06685=1072.928,39.181,434.853,173.163,23.889,154.263
C06686=1072.922,38.931,434.869,173.162,23.887,154.263
C06687=1072.916,38.682,434.886,173.161,23.884,154.262
C06688=1072.911,38.433,434.901,173.159,23.882,154.262
C06689=1072.905,38.183,434.917,173.158,23.879,154.262
C06690=1072.899,37.933,434.933,173.156,23.876,154.261
C06691=1072.892,37.684,434.948,173.154,23.873,154.261
C06692=1072.887,37.435,434.964,173.153,23.871,154.261
C06693=1072.881,37.185,434.980,173.152,23.868,154.260
C06694=1072.874,36.936,434.996,173.151,23.866,154.260
C06695=1072.869,36.687,435.011,173.149,23.863,154.260
C06696=1072.863,36.437,435.027,173.148,23.861,154.259
C06697=1072.858,36.187,435.043,173.147,23.858,154.259
C06698=1072.851,35.938,435.058,173.145,23.855,154.259
C06699=1072.845,35.688,435.074,173.143,23.853,154.258
C06700=1072.839,35.439,435.090,173.142,23.850,154.258
C06701=1072.834,35.190,435.105,173.141,23.848,154.258
C06702=1072.828,34.941,435.121,173.139,23.845,154.258
C06703=1072.822,34.691,435.137,173.138,23.843,154.257
C06704=1072.815,34.442,435.152,173.137,23.840,154.257
C06705=1072.810,34.192,435.168,173.136,23.837,154.257
C06706=1072.804,33.943,435.184,173.133,23.835,154.256
C06707=1072.799,33.693,435.199,173.132,23.832,154.256
C06708=1072.792,33.444,435.215,173.131,23.829,154.256
C06709=1072.786,33.194,435.230,173.130,23.827,154.255
C06710=1072.781,32.945,435.246,173.128,23.824,154.255
C06711=1072.775,32.696,435.261,173.127,23.822,154.255
C06712=1072.769,32.446,435.277,173.126,23.819,154.254
C06713=1072.763,32.197,435.293,173.124,23.817,154.254
C06714=1072.757,31.947,435.308,173.123,23.814,154.254
C06715=1072.751,31.698,435.323,173.121,23.811,154.253
C06716=1072.746,31.448,435.339,173.120,23.809,154.253
C06717=1072.739,31.199,435.354,173.118,23.806,154.253
C06718=1072.733,30.917,435.372,173.117,23.803,154.252
C06719=1072.726,30.635,435.389,173.115,23.800,154.252
C06720=1072.720,30.353,435.407,173.114,23.797,154.252
C06721=1072.713,30.071,435.424,173.113,23.794,154.251
C06722=1072.707,29.821,435.440,173.110,23.791,154.251
C06723=1072.701,29.571,435.456,173.109,23.789,154.251
C06724=1072.695,29.323,435.471,173.108,23.786,154.250
C06725=1072.690,29.073,435.486,173.107,23.784,154.250
C06726=1072.684,28.823,435.502,173.105,23.781,154.250
C06727=1072.678,28.573,435.517,173.104,23.779,154.249
C06728=1072.672,28.325,435.533,173.103,23.776,154.249
C06729=1072.666,28.075,435.548,173.102,23.774,154.249
C06730=1072.660,27.825,435.563,173.100,23.771,154.248
C06731=1072.654,27.577,435.579,173.098,23.768,154.248
C06732=1072.648,27.327,435.594,173.097,23.765,154.248
C06733=1072.642,27.077,435.609,173.095,23.763,154.248
C06734=1072.636,26.827,435.625,173.094,23.761,154.247
C06735=1072.630,26.579,435.640,173.093,23.758,154.247
C06736=1072.625,26.329,435.655,173.092,23.755,154.247
C06737=1072.618,26.079,435.670,173.090,23.753,154.246
C06738=1072.613,25.830,435.685,173.089,23.750,154.246
C06739=1072.607,25.580,435.700,173.087,23.748,154.246
C06740=1072.600,25.331,435.716,173.086,23.745,154.245
C06741=1072.595,25.082,435.731,173.084,23.742,154.245
C06742=1072.589,24.832,435.746,173.083,23.740,154.245
C06743=1072.583,24.582,435.762,173.082,23.738,154.244
C06744=1072.577,24.333,435.777,173.081,23.735,154.244
C06745=1072.572,24.084,435.792,173.079,23.732,154.244
C06746=1072.565,23.834,435.807,173.078,23.730,154.244
C06747=1072.559,23.585,435.823,173.077,23.727,154.243
C06748=1072.554,23.336,435.838,173.074,23.724,154.243
C06749=1072.547,23.086,435.853,173.073,23.722,154.243
C06750=1072.542,22.836,435.868,173.072,23.719,154.242
C06751=1072.536,22.587,435.883,173.071,23.717,154.242
C06752=1072.530,22.337,435.898,173.069,23.714,154.242
C06753=1072.524,22.088,435.913,173.068,23.712,154.241
C06754=1072.518,21.838,435.928,173.067,23.709,154.241
C06755=1072.512,21.588,435.943,173.065,23.707,154.241
C06756=1072.506,21.340,435.958,173.064,23.704,154.240
C06757=1072.501,21.090,435.974,173.063,23.701,154.240
C06758=1072.494,20.840,435.989,173.061,23.699,154.240
C06759=1072.488,20.592,436.004,173.059,23.696,154.240
C06760=1072.483,20.342,436.019,173.058,23.693,154.239
C06761=1072.477,20.093,436.034,173.057,23.691,154.239
C06762=1072.471,19.843,436.049,173.056,23.688,154.239
C06763=1072.465,19.593,436.064,173.054,23.686,154.238
C06764=1072.459,19.344,436.079,173.053,23.683,154.238
C06765=1072.453,19.094,436.094,173.052,23.681,154.238
C06766=1072.448,18.845,436.109,173.050,23.678,154.237
C06767=1072.441,18.595,436.124,173.048,23.676,154.237
C06768=1072.435,18.346,436.139,173.047,23.673,154.237
C06769=1072.429,18.097,436.153,173.046,23.670,154.236
C06770=1072.424,17.847,436.169,173.044,23.668,154.236
C06771=1072.418,17.597,436.183,173.043,23.665,154.236
C06772=1072.412,17.348,436.198,173.042,23.663,154.236
C06773=1072.406,17.098,436.213,173.040,23.661,154.235
C06774=1072.400,16.849,436.228,173.039,23.658,154.235
C06775=1072.394,16.599,436.243,173.038,23.655,154.235
C06776=1072.388,16.350,436.257,173.036,23.652,154.234
C06777=1072.382,16.100,436.273,173.034,23.650,154.234
C06778=1072.377,15.851,436.288,173.033,23.648,154.234
C06779=1072.370,15.602,436.303,173.032,23.645,154.233
C06780=1072.364,15.352,436.317,173.031,23.642,154.233
C06781=1072.359,15.103,436.333,173.029,23.640,154.233
C06782=1072.352,14.821,436.348,173.028,23.637,154.232
C06783=1072.345,14.541,436.365,173.026,23.634,154.232
C06784=1072.338,14.260,436.382,173.025,23.631,154.232
C06785=1072.332,13.980,436.399,173.023,23.628,154.231
C06786=1072.326,13.730,436.414,173.021,23.626,154.231
C06787=1072.320,13.481,436.428,173.020,23.624,154.231
C06788=1072.314,13.231,436.442,173.019,23.621,154.230
C06789=1072.308,12.982,436.457,173.018,23.618,154.230
C06790=1072.302,12.733,436.472,173.016,23.616,154.230
C06791=1072.295,12.483,436.487,173.015,23.613,154.230
C06792=1072.290,12.234,436.501,173.014,23.611,154.229
C06793=1072.284,11.984,436.516,173.012,23.609,154.229
C06794=1072.277,11.734,436.531,173.011,23.606,154.229
C06795=1072.271,11.485,436.545,173.009,23.603,154.229
C06796=1072.265,11.235,436.560,173.007,23.601,154.228
C06797=1072.260,10.986,436.574,173.006,23.598,154.228
C06798=1072.253,10.736,436.589,173.005,23.596,154.228
C06799=1072.247,10.487,436.603,173.004,23.593,154.227
C06800=1072.241,10.237,436.618,173.002,23.591,154.227
C06801=1072.236,9.988,436.632,173.001,23.588,154.227
C06802=1072.230,9.738,436.648,173.000,23.586,154.226
C06803=1072.224,9.489,436.662,172.998,23.584,154.226
C06804=1072.218,9.239,436.677,172.997,23.581,154.226
C06805=1072.212,8.990,436.691,172.995,23.578,154.226
C06806=1072.206,8.740,436.706,172.994,23.576,154.225
C06807=1072.200,8.491,436.720,172.992,23.573,154.225
C06808=1072.194,8.241,436.735,172.991,23.571,154.225
C06809=1072.188,7.992,436.750,172.990,23.568,154.224
C06810=1072.182,7.742,436.764,172.988,23.566,154.224
C06811=1072.176,7.493,436.778,172.987,23.563,154.224
C06812=1072.170,7.243,436.793,172.986,23.561,154.224
C06813=1072.165,6.994,436.807,172.985,23.559,154.223
C06814=1072.158,6.744,436.822,172.983,23.556,154.223
C06815=1072.152,6.495,436.835,172.981,23.553,154.223
C06816=1072.146,6.245,436.850,172.980,23.550,154.222
C06817=1072.140,5.995,436.864,172.979,23.548,154.222
C06818=1072.134,5.746,436.879,172.977,23.546,154.222
C06819=1072.128,5.497,436.894,172.976,23.543,154.222
C06820=1072.122,5.247,436.908,172.975,23.541,154.221
C06821=1072.116,4.998,436.923,172.973,23.538,154.221
C06822=1072.111,4.748,436.936,172.972,23.536,154.221
C06823=1072.104,4.498,436.951,172.971,23.534,154.220
C06824=1072.099,4.249,436.965,172.969,23.531,154.220
C06825=1072.093,4.000,436.980,172.967,23.528,154.220
C06826=1072.087,3.750,436.994,172.966,23.525,154.219
C06827=1072.081,3.501,437.009,172.965,23.523,154.219
C06828=1072.075,3.250,437.023,172.963,23.521,154.219
C06829=1072.069,3.001,437.037,172.962,23.518,154.219
C06830=1072.064,2.752,437.051,172.961,23.516,154.218
C06831=1072.057,2.502,437.066,172.960,23.513,154.218
C06832=1072.052,2.253,437.080,172.958,23.511,154.218
C06833=1072.046,2.004,437.095,172.957,23.508,154.217
C06834=1072.040,1.753,437.109,172.956,23.506,154.217
C06835=1072.034,1.504,437.124,172.953,23.503,154.217
C06836=1072.028,1.255,437.137,172.952,23.500,154.217
C06837=1072.022,1.005,437.152,172.951,23.498,154.216
C06838=1072.016,0.756,437.166,172.950,23.495,154.216
C06839=1072.010,0.506,437.180,172.948,23.493,154.216
C06840=1072.004,0.257,437.194,172.947,23.491,154.215
C06841=1071.999,0.007,437.208,172.946,23.488,154.215
C06842=1071.992,-0.243,437.223,172.944,23.486,154.215
C06843=1071.987,-0.492,437.237,172.943,23.483,154.215
C06844=1071.982,-0.742,437.251,172.942,23.481,154.214
C06845=1071.976,-0.991,437.266,172.940,23.478,154.214
C06846=1071.968,-1.304,437.283,172.938,23.475,154.214
C06847=1071.961,-1.617,437.301,172.936,23.472,154.213
C06848=1071.953,-1.931,437.319,172.935,23.469,154.213
C06849=1071.946,-2.243,437.336,172.933,23.466,154.213
C06850=1071.940,-2.492,437.350,172.932,23.463,154.212
C06851=1071.934,-2.742,437.365,172.931,23.461,154.212
C06852=1071.928,-2.992,437.379,172.929,23.458,154.212
C06853=1071.923,-3.241,437.392,172.928,23.456,154.211
C06854=1071.916,-3.491,437.407,172.926,23.453,154.211
C06855=1071.910,-3.740,437.421,172.925,23.451,154.211
C06856=1071.905,-3.990,437.435,172.923,23.448,154.211
C06857=1071.899,-4.240,437.449,172.922,23.446,154.210
C06858=1071.892,-4.489,437.463,172.921,23.443,154.210
C06859=1071.887,-4.738,437.477,172.919,23.441,154.210
C06860=1071.881,-4.988,437.491,172.918,23.439,154.209
C06861=1071.874,-5.238,437.504,172.917,23.436,154.209
C06862=1071.869,-5.487,437.519,172.915,23.434,154.209
C06863=1071.862,-5.737,437.532,172.914,23.431,154.209
C06864=1071.856,-5.986,437.546,172.913,23.429,154.208
C06865=1071.851,-6.236,437.560,172.911,23.426,154.208
C06866=1071.844,-6.486,437.574,172.909,23.424,154.208
C06867=1071.838,-6.735,437.588,172.908,23.421,154.208
C06868=1071.833,-6.984,437.602,172.907,23.419,154.207
C06869=1071.827,-7.234,437.615,172.905,23.417,154.207
C06870=1071.821,-7.484,437.630,172.904,23.415,154.207
C06871=1071.814,-7.733,437.643,172.903,23.412,154.207
C06872=1071.809,-7.983,437.657,172.901,23.410,154.206
C06873=1071.802,-8.232,437.672,172.900,23.407,154.206
C06874=1071.796,-8.482,437.685,172.899,23.405,154.206
C06875=1071.791,-8.731,437.699,172.897,23.402,154.205
C06876=1071.785,-8.980,437.712,172.895,23.400,154.205
C06877=1071.778,-9.231,437.726,172.894,23.397,154.205
C06878=1071.773,-9.480,437.740,172.893,23.395,154.205
C06879=1071.767,-9.729,437.754,172.891,23.392,154.204
C06880=1071.761,-9.979,437.767,172.890,23.390,154.204
C06881=1071.754,-10.228,437.782,172.889,23.388,154.204
C06882=1071.749,-10.478,437.796,172.887,23.385,154.204
C06883=1071.742,-10.727,437.809,172.886,23.383,154.203
C06884=1071.737,-10.977,437.823,172.885,23.381,154.203
C06885=1071.732,-11.226,437.837,172.883,23.378,154.203
C06886=1071.725,-11.476,437.850,172.881,23.376,154.203
C06887=1071.719,-11.726,437.864,172.880,23.373,154.202
C06888=1071.713,-11.975,437.877,172.879,23.371,154.202
C06889=1071.708,-12.225,437.891,172.877,23.368,154.202
C06890=1071.701,-12.474,437.905,172.876,23.366,154.201
C06891=1071.695,-12.724,437.919,172.875,23.364,154.201
C06892=1071.689,-12.974,437.932,172.873,23.361,154.201
C06893=1071.684,-13.223,437.946,172.872,23.359,154.201
C06894=1071.677,-13.472,437.959,172.871,23.356,154.200
C06895=1071.672,-13.722,437.973,172.869,23.354,154.200
C06896=1071.666,-13.972,437.987,172.867,23.352,154.200
C06897=1071.660,-14.222,438.000,172.866,23.349,154.200
C06898=1071.654,-14.454,438.013,172.865,23.347,154.199
C06899=1071.649,-14.686,438.026,172.863,23.344,154.199
C06900=1071.643,-14.919,438.039,172.863,23.343,154.199
C06901=1071.637,-15.151,438.051,172.861,23.340,154.199
C06902=1071.632,-15.384,438.063,172.860,23.338,154.198
C06903=1071.627,-15.616,438.076,172.859,23.336,154.198
C06904=1071.622,-15.848,438.089,172.857,23.334,154.198
C06905=1071.615,-16.081,438.101,172.856,23.332,154.198
C06906=1071.610,-16.330,438.115,172.855,23.329,154.197
C06907=1071.603,-16.580,438.128,172.853,23.327,154.197
C06908=1071.597,-16.829,438.142,172.852,23.325,154.197
C06909=1071.592,-17.079,438.155,172.850,23.322,154.197
C06910=1071.584,-17.356,438.170,172.849,23.319,154.196
C06911=1071.577,-17.633,438.184,172.847,23.317,154.196
C06912=1071.572,-17.910,438.200,172.845,23.314,154.196
C06913=1071.564,-18.187,438.214,172.844,23.312,154.196
C06914=1071.558,-18.436,438.228,172.842,23.309,154.195
C06915=1071.553,-18.686,438.242,172.841,23.307,154.195
C06916=1071.546,-18.935,438.255,172.840,23.305,154.195
C06917=1071.540,-19.185,438.268,172.838,23.303,154.195
C06918=1071.534,-19.435,438.282,172.837,23.300,154.194
C06919=1071.528,-19.685,438.295,172.836,23.298,154.194
C06920=1071.522,-19.934,438.308,172.833,23.295,154.194
C06921=1071.517,-20.184,438.322,172.832,23.293,154.194
C06922=1071.511,-20.433,438.335,172.831,23.291,154.193
C06923=1071.504,-20.683,438.348,172.830,23.288,154.193
C06924=1071.499,-20.932,438.362,172.828,23.286,154.193
C06925=1071.492,-21.182,438.375,172.827,23.284,154.193
C06926=1071.486,-21.432,438.388,172.826,23.281,154.192
C06927=1071.480,-21.681,438.401,172.824,23.279,154.192
C06928=1071.475,-21.931,438.415,172.823,23.277,154.192
C06929=1071.468,-22.180,438.428,172.821,23.275,154.192
C06930=1071.462,-22.430,438.441,172.820,23.272,154.191
C06931=1071.457,-22.680,438.455,172.818,23.269,154.191
C06932=1071.451,-22.929,438.468,172.817,23.268,154.191
C06933=1071.445,-23.178,438.481,172.815,23.265,154.191
C06934=1071.439,-23.428,438.494,172.814,23.263,154.190
C06935=1071.433,-23.678,438.508,172.813,23.260,154.190
C06936=1071.427,-23.927,438.521,172.811,23.258,154.190
C06937=1071.421,-24.177,438.534,172.810,23.256,154.190
C06938=1071.415,-24.426,438.547,172.809,23.254,154.189
C06939=1071.409,-24.676,438.561,172.807,23.251,154.189
C06940=1071.403,-24.926,438.573,172.806,23.249,154.189
C06941=1071.397,-25.175,438.586,172.805,23.247,154.189
C06942=1071.391,-25.425,438.599,172.803,23.244,154.188
C06943=1071.385,-25.675,438.613,172.801,23.242,154.188
C06944=1071.379,-25.924,438.627,172.800,23.240,154.188
C06945=1071.373,-26.174,438.639,172.798,23.237,154.188
C06946=1071.367,-26.423,438.652,172.797,23.235,154.188
C06947=1071.362,-26.674,438.665,172.796,23.233,154.187
C06948=1071.356,-26.923,438.679,172.794,23.231,154.187
C06949=1071.349,-27.172,438.692,172.793,23.228,154.187
C06950=1071.343,-27.422,438.705,172.792,23.226,154.187
C06951=1071.337,-27.671,438.718,172.790,23.224,154.186
C06952=1071.331,-27.921,438.730,172.789,23.221,154.186
C06953=1071.325,-28.170,438.744,172.788,23.220,154.186
C06954=1071.319,-28.420,438.756,172.785,23.217,154.186
C06955=1071.313,-28.670,438.770,172.784,23.215,154.186
C06956=1071.307,-28.919,438.782,172.783,23.212,154.185
C06957=1071.301,-29.169,438.795,172.781,23.210,154.185
C06958=1071.295,-29.419,438.808,172.780,23.208,154.185
C06959=1071.289,-29.668,438.821,172.779,23.206,154.185
C06960=1071.283,-29.918,438.834,172.777,23.204,154.184
C06961=1071.277,-30.167,438.847,172.776,23.201,154.184
C06962=1071.271,-30.417,438.860,172.774,23.199,154.184
C06963=1071.264,-30.666,438.873,172.773,23.197,154.184
C06964=1071.259,-30.916,438.885,172.772,23.195,154.183
C06965=1071.252,-31.165,438.899,172.769,23.192,154.183
C06966=1071.246,-31.415,438.911,172.768,23.190,154.183
C06967=1071.240,-31.664,438.924,172.767,23.188,154.183
C06968=1071.234,-31.914,438.937,172.765,23.186,154.183
C06969=1071.228,-32.164,438.950,172.764,23.184,154.183
C06970=1071.222,-32.413,438.963,172.763,23.181,154.182
C06971=1071.216,-32.663,438.975,172.761,23.179,154.182
C06972=1071.210,-32.913,438.989,172.760,23.177,154.182
C06973=1071.204,-33.162,439.001,172.759,23.175,154.182
C06974=1071.198,-33.438,439.015,172.756,23.172,154.181
C06975=1071.192,-33.714,439.030,172.755,23.170,154.181
C06976=1071.185,-33.991,439.044,172.754,23.167,154.181
C06977=1071.178,-34.268,439.058,172.752,23.165,154.181
C06978=1071.172,-34.517,439.071,172.750,23.162,154.180
C06979=1071.166,-34.767,439.083,172.749,23.160,154.180
C06980=1071.160,-35.017,439.096,172.748,23.158,154.180
C06981=1071.154,-35.265,439.109,172.746,23.156,154.180
C06982=1071.148,-35.515,439.121,172.745,23.154,154.179
C06983=1071.142,-35.765,439.134,172.743,23.152,154.179
C06984=1071.136,-36.014,439.147,172.742,23.149,154.179
C06985=1071.130,-36.264,439.160,172.741,23.147,154.179
C06986=1071.124,-36.514,439.172,172.739,23.145,154.179
C06987=1071.118,-36.764,439.185,172.738,23.143,154.178
C06988=1071.112,-37.013,439.198,172.737,23.141,154.178
C06989=1071.106,-37.263,439.211,172.735,23.139,154.178
C06990=1071.101,-37.512,439.223,172.733,23.136,154.178
C06991=1071.095,-37.761,439.236,172.732,23.134,154.178
C06992=1071.089,-38.011,439.249,172.730,23.132,154.177
C06993=1071.083,-38.261,439.261,172.729,23.130,154.177
C06994=1071.077,-38.511,439.274,172.727,23.127,154.177
C06995=1071.070,-38.761,439.286,172.726,23.125,154.177
C06996=1071.064,-39.010,439.299,172.725,23.123,154.177
C06997=1071.059,-39.259,439.311,172.723,23.121,154.176
C06998=1071.053,-39.509,439.324,172.722,23.119,154.176
C06999=1071.046,-39.759,439.336,172.721,23.117,154.176
C07000=1071.040,-40.008,439.348,172.719,23.115,154.176
C07001=1071.034,-40.258,439.362,172.718,23.112,154.176
C07002=1071.028,-40.508,439.374,172.715,23.110,154.175
C07003=1071.022,-40.757,439.386,172.714,23.108,154.175
C07004=1071.016,-41.007,439.399,172.713,23.106,154.175
C07005=1071.010,-41.257,439.411,172.711,23.104,154.175
C07006=1071.005,-41.506,439.423,172.710,23.102,154.175
C07007=1070.998,-41.755,439.436,172.709,23.100,154.174
C07008=1070.992,-42.005,439.449,172.707,23.098,154.174
C07009=1070.986,-42.255,439.461,172.706,23.095,154.174
C07010=1070.980,-42.505,439.474,172.704,23.093,154.174
C07011=1070.973,-42.754,439.486,172.703,23.092,154.174
C07012=1070.968,-43.003,439.498,172.702,23.089,154.173
C07013=1070.962,-43.253,439.510,172.700,23.087,154.173
C07014=1070.956,-43.503,439.523,172.699,23.085,154.173
C07015=1070.949,-43.753,439.535,172.697,23.082,154.173
C07016=1070.944,-44.003,439.547,172.695,23.081,154.173
C07017=1070.938,-44.253,439.560,172.694,23.079,154.173
C07018=1070.931,-44.501,439.572,172.692,23.076,154.172
C07019=1070.925,-44.751,439.585,172.691,23.074,154.172
C07020=1070.919,-45.001,439.597,172.690,23.073,154.172
C07021=1070.913,-45.250,439.609,172.688,23.070,154.172
C07022=1070.907,-45.500,439.622,172.687,23.068,154.172
C07023=1070.902,-45.749,439.634,172.685,23.066,154.171
C07024=1070.896,-45.999,439.647,172.684,23.064,154.171
C07025=1070.889,-46.249,439.659,172.683,23.062,154.171
C07026=1070.883,-46.499,439.671,172.681,23.060,154.171
C07027=1070.878,-46.748,439.683,172.679,23.058,154.171
C07028=1070.871,-46.997,439.695,172.678,23.055,154.170
C07029=1070.865,-47.247,439.708,172.676,23.054,154.170
C07030=1070.859,-47.497,439.720,172.675,23.052,154.170
C07031=1070.853,-47.746,439.732,172.673,23.049,154.170
C07032=1070.848,-47.996,439.744,172.672,23.047,154.170
C07033=1070.842,-48.246,439.756,172.670,23.045,154.170
C07034=1070.835,-48.496,439.768,172.669,23.044,154.169
C07035=1070.830,-48.745,439.781,172.668,23.041,154.169
C07036=1070.824,-48.995,439.793,172.666,23.039,154.169
C07037=1070.817,-49.245,439.805,172.665,23.037,154.169
C07038=1070.811,-49.522,439.819,172.663,23.034,154.169
C07039=1070.805,-49.798,439.832,172.661,23.033,154.169
C07040=1070.798,-50.075,439.846,172.660,23.030,154.168
C07041=1070.791,-50.351,439.859,172.658,23.028,154.168
C07042=1070.785,-50.601,439.871,172.656,23.026,154.168
C07043=1070.779,-50.851,439.883,172.655,23.024,154.168
C07044=1070.773,-51.100,439.895,172.653,23.022,154.168
C07045=1070.767,-51.349,439.907,172.652,23.020,154.167
C07046=1070.760,-51.599,439.919,172.651,23.018,154.167
C07047=1070.753,-51.849,439.931,172.649,23.016,154.167
C07048=1070.748,-52.098,439.943,172.648,23.014,154.167
C07049=1070.742,-52.348,439.955,172.646,23.012,154.167
C07050=1070.736,-52.598,439.967,172.645,23.010,154.167
C07051=1070.729,-52.847,439.979,172.643,23.008,154.167
C07052=1070.723,-53.096,439.991,172.642,23.007,154.166
C07053=1070.718,-53.347,440.003,172.640,23.005,154.166
C07054=1070.711,-53.596,440.015,172.639,23.003,154.166
C07055=1070.704,-53.846,440.027,172.637,23.001,154.166
C07056=1070.699,-54.095,440.039,172.635,22.999,154.166
C07057=1070.693,-54.345,440.050,172.634,22.997,154.166
C07058=1070.686,-54.595,440.062,172.632,22.995,154.166
C07059=1070.680,-54.845,440.075,172.631,22.993,154.165
C07060=1070.674,-55.094,440.086,172.630,22.991,154.165
C07061=1070.668,-55.344,440.098,172.628,22.989,154.165
C07062=1070.662,-55.594,440.110,172.627,22.987,154.165
C07063=1070.656,-55.843,440.122,172.625,22.985,154.165
C07064=1070.650,-56.092,440.134,172.624,22.983,154.165
C07065=1070.643,-56.343,440.145,172.622,22.981,154.164
C07066=1070.637,-56.591,440.157,172.621,22.979,154.164
C07067=1070.631,-56.841,440.169,172.619,22.977,154.164
C07068=1070.625,-57.092,440.181,172.618,22.975,154.164
C07069=1070.619,-57.340,440.192,172.617,22.974,154.164
C07070=1070.612,-57.590,440.204,172.615,22.972,154.164
C07071=1070.607,-57.841,440.216,172.613,22.969,154.164
C07072=1070.601,-58.089,440.228,172.611,22.967,154.163
C07073=1070.594,-58.339,440.240,172.610,22.966,154.163
C07074=1070.589,-58.589,440.252,172.608,22.964,154.163
C07075=1070.582,-58.838,440.263,172.607,22.962,154.163
C07076=1070.576,-59.089,440.274,172.606,22.960,154.163
C07077=1070.570,-59.338,440.287,172.604,22.958,154.163
C07078=1070.564,-59.587,440.299,172.602,22.957,154.163
C07079=1070.558,-59.837,440.310,172.601,22.955,154.162
C07080=1070.551,-60.087,440.322,172.600,22.953,154.162
C07081=1070.546,-60.337,440.333,172.598,22.951,154.162
C07082=1070.540,-60.586,440.345,172.597,22.949,154.162
C07083=1070.534,-60.835,440.357,172.595,22.947,154.162
C07084=1070.528,-61.086,440.369,172.594,22.945,154.162
C07085=1070.521,-61.335,440.381,172.592,22.943,154.162
C07086=1070.516,-61.585,440.391,172.590,22.941,154.161
C07087=1070.509,-61.834,440.403,172.589,22.939,154.161
C07088=1070.504,-62.084,440.415,172.587,22.937,154.161
C07089=1070.497,-62.334,440.427,172.586,22.935,154.161
C07090=1070.491,-62.584,440.438,172.584,22.934,154.161
C07091=1070.485,-62.833,440.450,172.583,22.932,154.161
C07092=1070.479,-63.083,440.461,172.581,22.930,154.161
C07093=1070.473,-63.332,440.473,172.580,22.928,154.160
C07094=1070.467,-63.582,440.484,172.578,22.927,154.160
C07095=1070.461,-63.831,440.496,172.577,22.925,154.160
C07096=1070.455,-64.082,440.508,172.575,22.923,154.160
C07097=1070.449,-64.331,440.519,172.574,22.921,154.160
C07098=1070.443,-64.581,440.531,172.572,22.919,154.160
C07099=1070.437,-64.830,440.542,172.571,22.917,154.160
C07100=1070.431,-65.080,440.554,172.570,22.915,154.160
C07101=1070.425,-65.330,440.566,172.568,22.913,154.159
C07102=1070.418,-65.608,440.578,172.566,22.911,154.159
C07103=1070.411,-65.886,440.591,172.564,22.909,154.159
C07104=1070.405,-66.163,440.604,172.563,22.907,154.159
C07105=1070.398,-66.442,440.617,172.561,22.905,154.159
C07106=1070.392,-66.691,440.628,172.559,22.903,154.159
C07107=1070.386,-66.941,440.640,172.558,22.901,154.159
C07108=1070.380,-67.190,440.651,172.556,22.899,154.158
C07109=1070.374,-67.440,440.662,172.555,22.898,154.158
C07110=1070.368,-67.690,440.674,172.553,22.896,154.158
C07111=1070.362,-67.940,440.686,172.552,22.894,154.158
C07112=1070.356,-68.189,440.696,172.550,22.892,154.158
C07113=1070.350,-68.439,440.708,172.549,22.890,154.158
C07114=1070.344,-68.688,440.719,172.547,22.889,154.158
C07115=1070.339,-68.938,440.731,172.546,22.887,154.158
C07116=1070.332,-69.188,440.743,172.544,22.885,154.158
C07117=1070.327,-69.437,440.754,172.543,22.883,154.157
C07118=1070.320,-69.687,440.765,172.541,22.882,154.157
C07119=1070.314,-69.936,440.776,172.540,22.880,154.157
C07120=1070.308,-70.187,440.788,172.538,22.878,154.157
C07121=1070.303,-70.436,440.799,172.537,22.876,154.157
C07122=1070.296,-70.686,440.811,172.536,22.874,154.157
C07123=1070.290,-70.935,440.822,172.534,22.873,154.157
C07124=1070.285,-71.185,440.833,172.532,22.870,154.157
C07125=1070.278,-71.435,440.844,172.530,22.869,154.157
C07126=1070.272,-71.684,440.856,172.529,22.867,154.156
C07127=1070.267,-71.934,440.867,172.527,22.865,154.156
C07128=1070.261,-72.184,440.878,172.526,22.863,154.156
C07129=1070.255,-72.433,440.889,172.524,22.862,154.156
C07130=1070.249,-72.683,440.901,172.523,22.860,154.156
C07131=1070.243,-72.932,440.912,172.521,22.858,154.156
C07132=1070.236,-73.183,440.923,172.520,22.856,154.156
C07133=1070.231,-73.432,440.934,172.518,22.855,154.156
C07134=1070.226,-73.682,440.946,172.517,22.853,154.155
C07135=1070.219,-73.932,440.958,172.515,22.851,154.155
C07136=1070.213,-74.181,440.969,172.514,22.849,154.155
C07137=1070.207,-74.431,440.980,172.512,22.848,154.155
C07138=1070.201,-74.681,440.991,172.511,22.846,154.155
C07139=1070.196,-74.930,441.002,172.509,22.845,154.155
C07140=1070.189,-75.180,441.013,172.508,22.843,154.155
C07141=1070.183,-75.430,441.023,172.506,22.841,154.155
C07142=1070.176,-75.679,441.035,172.505,22.840,154.155
C07143=1070.170,-75.929,441.046,172.503,22.838,154.155
C07144=1070.165,-76.178,441.057,172.502,22.836,154.155
C07145=1070.158,-76.428,441.068,172.500,22.834,154.154
C07146=1070.152,-76.678,441.079,172.499,22.833,154.154
C07147=1070.146,-76.928,441.090,172.496,22.831,154.154
C07148=1070.140,-77.177,441.101,172.495,22.829,154.154
C07149=1070.135,-77.427,441.112,172.493,22.828,154.154
C07150=1070.128,-77.677,441.123,172.492,22.826,154.154
C07151=1070.123,-77.927,441.134,172.490,22.824,154.154
C07152=1070.116,-78.176,441.146,172.489,22.822,154.154
C07153=1070.109,-78.425,441.156,172.487,22.821,154.154
C07154=1070.104,-78.675,441.167,172.486,22.819,154.154
C07155=1070.097,-78.925,441.178,172.484,22.818,154.154
C07156=1070.092,-79.175,441.189,172.483,22.816,154.153
C07157=1070.086,-79.424,441.200,172.481,22.815,154.153
C07158=1070.080,-79.674,441.211,172.480,22.813,154.153
C07159=1070.074,-79.924,441.222,172.478,22.811,154.153
C07160=1070.067,-80.173,441.233,172.477,22.809,154.153
C07161=1070.061,-80.423,441.244,172.475,22.808,154.153
C07162=1070.055,-80.673,441.255,172.473,22.807,154.153
C07163=1070.049,-80.923,441.266,172.472,22.805,154.153
C07164=1070.042,-81.172,441.276,172.470,22.804,154.153
C07165=1070.037,-81.421,441.287,172.469,22.802,154.153
C07166=1070.030,-81.702,441.299,172.467,22.800,154.153
C07167=1070.023,-81.982,441.311,172.465,22.798,154.153
C07168=1070.016,-82.262,441.324,172.463,22.797,154.153
C07169=1070.009,-82.542,441.335,172.462,22.795,154.153
C07170=1070.003,-82.792,441.347,172.460,22.793,154.152
C07171=1069.997,-83.042,441.358,172.459,22.792,154.152
C07172=1069.990,-83.291,441.368,172.457,22.790,154.152
C07173=1069.984,-83.542,441.378,172.456,22.789,154.152
C07174=1069.979,-83.791,441.389,172.454,22.788,154.152
C07175=1069.972,-84.040,441.399,172.452,22.786,154.152
C07176=1069.966,-84.291,441.411,172.451,22.784,154.152
C07177=1069.960,-84.540,441.422,172.449,22.783,154.152
C07178=1069.954,-84.789,441.432,172.448,22.781,154.152
C07179=1069.947,-85.039,441.443,172.445,22.779,154.152
C07180=1069.941,-85.289,441.454,172.444,22.778,154.152
C07181=1069.935,-85.539,441.464,172.442,22.777,154.152
C07182=1069.929,-85.789,441.475,172.441,22.775,154.152
C07183=1069.923,-86.038,441.486,172.439,22.773,154.152
C07184=1069.917,-86.288,441.496,172.437,22.772,154.152
C07185=1069.911,-86.537,441.507,172.436,22.770,154.152
C07186=1069.904,-86.787,441.517,172.434,22.769,154.152
C07187=1069.898,-87.037,441.528,172.433,22.768,154.152
C07188=1069.893,-87.287,441.539,172.431,22.766,154.152
C07189=1069.886,-87.536,441.549,172.430,22.764,154.151
C07190=1069.880,-87.786,441.560,172.428,22.763,154.151
C07191=1069.874,-88.035,441.571,172.426,22.762,154.151
C07192=1069.868,-88.285,441.581,172.425,22.760,154.151
C07193=1069.862,-88.535,441.592,172.423,22.758,154.151
C07194=1069.856,-88.785,441.603,172.422,22.757,154.151
C07195=1069.849,-89.034,441.613,172.420,22.756,154.151
C07196=1069.844,-89.284,441.623,172.419,22.754,154.151
C07197=1069.837,-89.534,441.634,172.417,22.753,154.151
C07198=1069.831,-89.784,441.645,172.416,22.751,154.151
C07199=1069.825,-90.033,441.655,172.414,22.750,154.151
C07200=1069.819,-90.283,441.665,172.412,22.748,154.151
C07201=1069.814,-90.532,441.676,172.411,22.747,154.151
C07202=1069.806,-90.782,441.687,172.409,22.746,154.151
C07203=1069.801,-91.032,441.697,172.408,22.744,154.151
C07204=1069.795,-91.282,441.708,172.406,22.742,154.151
C07205=1069.789,-91.531,441.718,172.404,22.741,154.151
C07206=1069.783,-91.781,441.728,172.403,22.740,154.151
C07207=1069.776,-92.031,441.739,172.401,22.738,154.151
C07208=1069.771,-92.280,441.750,172.400,22.737,154.151
C07209=1069.765,-92.531,441.760,172.398,22.735,154.151
C07210=1069.759,-92.780,441.770,172.396,22.734,154.151
C07211=1069.753,-93.029,441.781,172.395,22.733,154.151
C07212=1069.747,-93.279,441.790,172.393,22.731,154.151
C07213=1069.740,-93.529,441.802,172.392,22.730,154.151
C07214=1069.734,-93.779,441.811,172.390,22.729,154.151
C07215=1069.728,-94.029,441.822,172.388,22.727,154.151
C07216=1069.723,-94.278,441.833,172.387,22.725,154.150
C07217=1069.717,-94.528,441.843,172.385,22.724,154.150
C07218=1069.711,-94.777,441.853,172.384,22.723,154.150
C07219=1069.704,-95.028,441.863,172.382,22.721,154.150
C07220=1069.698,-95.277,441.874,172.381,22.720,154.150
C07221=1069.692,-95.526,441.885,172.379,22.719,154.150
C07222=1069.686,-95.777,441.895,172.377,22.717,154.150
C07223=1069.680,-96.026,441.905,172.376,22.716,154.150
C07224=1069.674,-96.276,441.915,172.374,22.715,154.150
C07225=1069.669,-96.525,441.926,172.372,22.713,154.150
C07226=1069.663,-96.775,441.936,172.371,22.712,154.150
C07227=1069.657,-97.025,441.946,172.369,22.710,154.150
C07228=1069.650,-97.275,441.956,172.368,22.709,154.150
C07229=1069.644,-97.525,441.967,172.366,22.707,154.150
C07230=1069.638,-97.807,441.979,172.365,22.706,154.150
C07231=1069.630,-98.090,441.990,172.362,22.704,154.150
C07232=1069.623,-98.372,442.001,172.360,22.703,154.150
C07233=1069.617,-98.654,442.012,172.359,22.702,154.150
C07234=1069.610,-98.903,442.023,172.357,22.700,154.150
C07235=1069.604,-99.154,442.033,172.356,22.699,154.150
C07236=1069.598,-99.403,442.043,172.354,22.698,154.150
C07237=1069.592,-99.653,442.053,172.352,22.697,154.150
C07238=1069.586,-99.903,442.064,172.351,22.695,154.150
C07239=1069.580,-100.152,442.073,172.349,22.694,154.150
C07240=1069.573,-100.402,442.084,172.347,22.693,154.150
C07241=1069.568,-100.652,442.094,172.346,22.691,154.150
C07242=1069.562,-100.901,442.103,172.344,22.690,154.150
C07243=1069.554,-101.151,442.114,172.343,22.689,154.150
C07244=1069.549,-101.401,442.124,172.341,22.688,154.150
C07245=1069.543,-101.651,442.135,172.339,22.687,154.150
C07246=1069.536,-101.900,442.144,172.337,22.685,154.150
C07247=1069.531,-102.151,442.154,172.336,22.684,154.150
C07248=1069.524,-102.400,442.165,172.334,22.683,154.150
C07249=1069.518,-102.650,442.174,172.333,22.681,154.150
C07250=1069.513,-102.899,442.185,172.331,22.680,154.150
C07251=1069.506,-103.149,442.195,172.329,22.679,154.150
C07252=1069.500,-103.399,442.204,172.328,22.678,154.150
C07253=1069.494,-103.648,442.214,172.326,22.676,154.150
C07254=1069.488,-103.898,442.225,172.324,22.675,154.150
C07255=1069.482,-104.148,442.234,172.323,22.674,154.150
C07256=1069.476,-104.397,442.244,172.321,22.673,154.150
C07257=1069.470,-104.648,442.255,172.319,22.672,154.150
C07258=1069.463,-104.897,442.265,172.318,22.670,154.150
C07259=1069.457,-105.147,442.274,172.316,22.669,154.150
C07260=1069.451,-105.396,442.284,172.314,22.668,154.150
C07261=1069.445,-105.647,442.295,172.313,22.667,154.150
C07262=1069.439,-105.896,442.304,172.311,22.665,154.150
C07263=1069.433,-106.146,442.314,172.310,22.664,154.150
C07264=1069.427,-106.395,442.324,172.308,22.663,154.150
C07265=1069.421,-106.645,442.334,172.306,22.662,154.150
C07266=1069.415,-106.895,442.344,172.305,22.661,154.150
C07267=1069.408,-107.144,442.354,172.303,22.660,154.150
C07268=1069.402,-107.394,442.364,172.302,22.659,154.150
C07269=1069.396,-107.644,442.373,172.300,22.658,154.150
C07270=1069.390,-107.894,442.383,172.299,22.657,154.150
C07271=1069.385,-108.144,442.393,172.297,22.655,154.150
C07272=1069.378,-108.393,442.403,172.295,22.654,154.150
C07273=1069.372,-108.643,442.413,172.294,22.653,154.151
C07274=1069.366,-108.893,442.422,172.292,22.652,154.151
C07275=1069.360,-109.142,442.432,172.290,22.651,154.150
C07276=1069.353,-109.392,442.441,172.289,22.650,154.151
C07277=1069.347,-109.642,442.451,172.287,22.648,154.151
C07278=1069.341,-109.891,442.461,172.285,22.648,154.151
C07279=1069.335,-110.141,442.471,172.284,22.646,154.151
C07280=1069.329,-110.391,442.481,172.282,22.646,154.151
C07281=1069.323,-110.641,442.491,172.280,22.644,154.151
C07282=1069.317,-110.891,442.500,172.279,22.643,154.151
C07283=1069.311,-111.141,442.510,172.277,22.642,154.151
